C01803=1094.320,109.025,-62.367,176.115,17.436,152.491
C01804=1094.315,108.775,-62.348,176.112,17.435,152.491
C01805=1094.309,108.526,-62.329,176.109,17.434,152.491
C01806=1094.303,108.277,-62.310,176.107,17.434,152.491
C01807=1094.297,108.028,-62.292,176.104,17.433,152.492
C01808=1094.292,107.779,-62.274,176.102,17.431,152.492
C01809=1094.287,107.529,-62.254,176.100,17.431,152.492
C01810=1094.280,107.279,-62.236,176.097,17.430,152.493
C01811=1094.275,107.031,-62.218,176.095,17.429,152.493
C01812=1094.269,106.782,-62.199,176.092,17.428,152.493
C01813=1094.264,106.532,-62.181,176.089,17.428,152.494
C01814=1094.258,106.283,-62.162,176.087,17.427,152.494
C01815=1094.253,106.034,-62.144,176.085,17.426,152.494
C01816=1094.247,105.785,-62.125,176.082,17.424,152.494
C01817=1094.241,105.535,-62.106,176.080,17.424,152.495
C01818=1094.236,105.286,-62.088,176.077,17.423,152.495
C01819=1094.230,105.037,-62.069,176.075,17.422,152.495
C01820=1094.225,104.787,-62.051,176.072,17.421,152.496
C01821=1094.218,104.538,-62.032,176.070,17.420,152.496
C01822=1094.214,104.289,-62.014,176.067,17.420,152.496
C01823=1094.207,104.040,-61.996,176.065,17.419,152.497
C01824=1094.202,103.790,-61.978,176.063,17.418,152.497
C01825=1094.196,103.541,-61.959,176.060,17.417,152.497
C01826=1094.191,103.292,-61.941,176.057,17.416,152.497
C01827=1094.185,103.043,-61.922,176.055,17.415,152.498
C01828=1094.180,102.794,-61.904,176.053,17.414,152.498
C01829=1094.174,102.544,-61.885,176.050,17.413,152.498
C01830=1094.169,102.295,-61.867,176.048,17.412,152.498
C01831=1094.162,102.046,-61.848,176.045,17.411,152.499
C01832=1094.158,101.797,-61.830,176.043,17.411,152.499
C01833=1094.152,101.547,-61.812,176.040,17.409,152.499
C01834=1094.146,101.298,-61.793,176.038,17.408,152.500
C01835=1094.140,101.048,-61.776,176.036,17.408,152.500
C01836=1094.134,100.800,-61.757,176.033,17.407,152.500
C01837=1094.129,100.550,-61.739,176.031,17.406,152.500
C01838=1094.124,100.301,-61.721,176.028,17.405,152.501
C01839=1094.117,100.052,-61.702,176.026,17.404,152.501
C01840=1094.112,99.802,-61.684,176.024,17.403,152.501
C01841=1094.106,99.553,-61.666,176.021,17.402,152.501
C01842=1094.100,99.304,-61.648,176.019,17.401,152.502
C01843=1094.095,99.054,-61.630,176.016,17.401,152.502
C01844=1094.090,98.805,-61.612,176.014,17.400,152.502
C01845=1094.083,98.556,-61.593,176.011,17.399,152.503
C01846=1094.078,98.307,-61.575,176.009,17.397,152.503
C01847=1094.072,98.057,-61.557,176.007,17.397,152.503
C01848=1094.066,97.809,-61.539,176.004,17.396,152.503
C01849=1094.060,97.559,-61.521,176.002,17.395,152.504
C01850=1094.055,97.309,-61.503,175.999,17.394,152.504
C01851=1094.049,97.060,-61.485,175.997,17.393,152.504
C01852=1094.044,96.811,-61.467,175.995,17.392,152.504
C01853=1094.039,96.562,-61.449,175.992,17.391,152.505
C01854=1094.033,96.312,-61.431,175.990,17.390,152.505
C01855=1094.026,96.037,-61.411,175.987,17.389,152.505
C01856=1094.020,95.761,-61.392,175.984,17.388,152.506
C01857=1094.014,95.485,-61.370,175.982,17.387,152.506
C01858=1094.008,95.210,-61.351,175.979,17.386,152.506
C01859=1094.002,94.961,-61.333,175.977,17.385,152.507
C01860=1093.996,94.711,-61.315,175.974,17.384,152.507
C01861=1093.991,94.462,-61.297,175.973,17.383,152.507
C01862=1093.985,94.213,-61.279,175.970,17.382,152.507
C01863=1093.979,93.963,-61.261,175.967,17.381,152.508
C01864=1093.974,93.714,-61.243,175.965,17.380,152.508
C01865=1093.969,93.465,-61.225,175.962,17.379,152.508
C01866=1093.963,93.215,-61.207,175.961,17.378,152.508
C01867=1093.957,92.966,-61.190,175.958,17.377,152.508
C01868=1093.951,92.716,-61.172,175.955,17.376,152.509
C01869=1093.946,92.467,-61.154,175.954,17.375,152.509
C01870=1093.941,92.218,-61.136,175.951,17.374,152.509
C01871=1093.935,91.968,-61.118,175.949,17.373,152.509
C01872=1093.929,91.719,-61.101,175.946,17.372,152.510
C01873=1093.923,91.471,-61.082,175.944,17.371,152.510
C01874=1093.917,91.221,-61.064,175.942,17.370,152.510
C01875=1093.912,90.972,-61.046,175.939,17.369,152.511
C01876=1093.907,90.723,-61.029,175.937,17.368,152.511
C01877=1093.901,90.473,-61.011,175.934,17.367,152.511
C01878=1093.895,90.224,-60.993,175.932,17.366,152.511
C01879=1093.890,89.975,-60.976,175.930,17.365,152.512
C01880=1093.884,89.725,-60.958,175.928,17.364,152.512
C01881=1093.878,89.476,-60.940,175.925,17.363,152.512
C01882=1093.873,89.227,-60.922,175.923,17.362,152.512
C01883=1093.866,88.977,-60.905,175.921,17.361,152.512
C01884=1093.861,88.728,-60.887,175.918,17.360,152.513
C01885=1093.856,88.479,-60.870,175.916,17.359,152.513
C01886=1093.850,88.229,-60.852,175.913,17.358,152.513
C01887=1093.844,87.980,-60.835,175.911,17.357,152.514
C01888=1093.839,87.731,-60.817,175.909,17.356,152.514
C01889=1093.832,87.481,-60.799,175.907,17.355,152.514
C01890=1093.827,87.232,-60.782,175.904,17.354,152.514
C01891=1093.821,86.983,-60.764,175.902,17.353,152.514
C01892=1093.815,86.733,-60.746,175.900,17.352,152.515
C01893=1093.810,86.484,-60.728,175.897,17.351,152.515
C01894=1093.804,86.235,-60.711,175.895,17.350,152.515
C01895=1093.798,85.985,-60.694,175.892,17.349,152.515
C01896=1093.793,85.736,-60.676,175.891,17.348,152.516
C01897=1093.787,85.487,-60.659,175.888,17.347,152.516
C01898=1093.781,85.238,-60.642,175.886,17.346,152.516
C01899=1093.775,84.988,-60.624,175.883,17.345,152.516
C01900=1093.770,84.739,-60.606,175.881,17.344,152.517
C01901=1093.764,84.490,-60.589,175.879,17.342,152.517
C01902=1093.759,84.241,-60.572,175.877,17.342,152.517
C01903=1093.753,83.991,-60.554,175.874,17.341,152.517
C01904=1093.747,83.742,-60.536,175.872,17.339,152.518
C01905=1093.742,83.492,-60.519,175.870,17.338,152.518
C01906=1093.736,83.243,-60.502,175.867,17.337,152.518
C01907=1093.730,82.993,-60.484,175.865,17.336,152.518
C01908=1093.725,82.744,-60.466,175.863,17.335,152.518
C01909=1093.720,82.495,-60.449,175.861,17.334,152.519
C01910=1093.714,82.246,-60.432,175.858,17.333,152.519
C01911=1093.708,81.997,-60.415,175.856,17.332,152.519
C01912=1093.702,81.746,-60.398,175.854,17.331,152.519
C01913=1093.696,81.497,-60.380,175.852,17.330,152.519
C01914=1093.691,81.248,-60.363,175.849,17.329,152.520
C01915=1093.685,80.999,-60.345,175.847,17.328,152.520
C01916=1093.680,80.750,-60.328,175.845,17.326,152.520
C01917=1093.675,80.501,-60.311,175.842,17.325,152.520
C01918=1093.669,80.250,-60.293,175.840,17.325,152.521
C01919=1093.662,79.975,-60.274,175.838,17.323,152.521
C01920=1093.656,79.700,-60.255,175.835,17.322,152.521
C01921=1093.650,79.424,-60.236,175.833,17.321,152.521
C01922=1093.644,79.149,-60.217,175.831,17.319,152.521
C01923=1093.639,78.900,-60.199,175.828,17.318,152.522
C01924=1093.633,78.650,-60.183,175.826,17.318,152.522
C01925=1093.627,78.400,-60.165,175.824,17.316,152.522
C01926=1093.621,78.151,-60.148,175.822,17.315,152.522
C01927=1093.616,77.902,-60.131,175.819,17.314,152.523
C01928=1093.610,77.652,-60.114,175.818,17.313,152.523
C01929=1093.604,77.403,-60.097,175.815,17.312,152.523
C01930=1093.599,77.154,-60.080,175.813,17.311,152.523
C01931=1093.592,76.904,-60.063,175.811,17.309,152.523
C01932=1093.587,76.655,-60.045,175.809,17.309,152.524
C01933=1093.582,76.406,-60.028,175.806,17.308,152.524
C01934=1093.576,76.157,-60.011,175.803,17.306,152.524
C01935=1093.570,75.907,-59.994,175.802,17.305,152.524
C01936=1093.565,75.658,-59.977,175.799,17.304,152.524
C01937=1093.559,75.409,-59.960,175.797,17.303,152.525
C01938=1093.553,75.158,-59.943,175.795,17.302,152.525
C01939=1093.547,74.909,-59.926,175.793,17.301,152.525
C01940=1093.541,74.660,-59.910,175.790,17.299,152.525
C01941=1093.536,74.411,-59.892,175.789,17.298,152.525
C01942=1093.531,74.161,-59.875,175.786,17.297,152.526
C01943=1093.524,73.913,-59.858,175.784,17.296,152.526
C01944=1093.519,73.663,-59.841,175.781,17.295,152.526
C01945=1093.514,73.414,-59.824,175.780,17.294,152.526
C01946=1093.508,73.165,-59.808,175.777,17.292,152.526
C01947=1093.502,72.914,-59.790,175.775,17.292,152.527
C01948=1093.496,72.665,-59.773,175.773,17.290,152.527
C01949=1093.490,72.416,-59.757,175.771,17.289,152.527
C01950=1093.485,72.166,-59.740,175.768,17.288,152.527
C01951=1093.479,71.917,-59.723,175.767,17.287,152.527
C01952=1093.474,71.668,-59.706,175.764,17.286,152.528
C01953=1093.468,71.418,-59.689,175.762,17.285,152.528
C01954=1093.462,71.169,-59.672,175.759,17.284,152.528
C01955=1093.457,70.920,-59.655,175.758,17.283,152.528
C01956=1093.451,70.670,-59.639,175.755,17.281,152.528
C01957=1093.446,70.421,-59.621,175.753,17.280,152.528
C01958=1093.440,70.172,-59.605,175.751,17.279,152.529
C01959=1093.434,69.922,-59.588,175.749,17.278,152.529
C01960=1093.429,69.673,-59.571,175.746,17.277,152.529
C01961=1093.423,69.424,-59.554,175.745,17.276,152.529
C01962=1093.417,69.175,-59.538,175.742,17.274,152.529
C01963=1093.412,68.925,-59.521,175.740,17.273,152.530
C01964=1093.405,68.676,-59.504,175.738,17.272,152.530
C01965=1093.400,68.426,-59.487,175.736,17.271,152.530
C01966=1093.394,68.177,-59.471,175.734,17.269,152.530
C01967=1093.388,67.927,-59.454,175.732,17.269,152.530
C01968=1093.383,67.677,-59.438,175.729,17.267,152.530
C01969=1093.377,67.428,-59.420,175.727,17.266,152.531
C01970=1093.371,67.179,-59.404,175.725,17.265,152.531
C01971=1093.366,66.929,-59.387,175.723,17.264,152.531
C01972=1093.360,66.680,-59.371,175.721,17.262,152.531
C01973=1093.355,66.430,-59.354,175.719,17.262,152.531
C01974=1093.348,66.182,-59.337,175.716,17.260,152.532
C01975=1093.342,65.932,-59.321,175.714,17.259,152.532
C01976=1093.337,65.683,-59.304,175.712,17.258,152.532
C01977=1093.331,65.433,-59.288,175.710,17.257,152.532
C01978=1093.326,65.184,-59.271,175.708,17.256,152.532
C01979=1093.320,64.934,-59.255,175.706,17.254,152.532
C01980=1093.314,64.685,-59.238,175.704,17.254,152.533
C01981=1093.309,64.435,-59.221,175.702,17.252,152.533
C01982=1093.303,64.186,-59.205,175.700,17.251,152.533
C01983=1093.297,63.911,-59.187,175.697,17.250,152.533
C01984=1093.290,63.636,-59.168,175.695,17.248,152.533
C01985=1093.283,63.360,-59.150,175.692,17.247,152.534
C01986=1093.277,63.085,-59.132,175.690,17.246,152.534
C01987=1093.272,62.835,-59.115,175.688,17.244,152.534
C01988=1093.266,62.586,-59.099,175.686,17.243,152.534
C01989=1093.260,62.336,-59.083,175.683,17.242,152.534
C01990=1093.254,62.087,-59.067,175.682,17.241,152.534
C01991=1093.249,61.837,-59.050,175.679,17.240,152.535
C01992=1093.243,61.588,-59.034,175.677,17.239,152.535
C01993=1093.237,61.339,-59.017,175.675,17.237,152.535
C01994=1093.231,61.089,-59.001,175.673,17.236,152.535
C01995=1093.225,60.840,-58.985,175.671,17.235,152.535
C01996=1093.220,60.590,-58.968,175.669,17.234,152.535
C01997=1093.214,60.341,-58.952,175.667,17.233,152.536
C01998=1093.208,60.092,-58.935,175.664,17.232,152.536
C01999=1093.202,59.842,-58.920,175.663,17.231,152.536
C02000=1093.196,59.592,-58.904,175.660,17.229,152.536
C02001=1093.191,59.343,-58.887,175.658,17.228,152.536
C02002=1093.185,59.093,-58.871,175.656,17.227,152.536
C02003=1093.179,58.844,-58.854,175.654,17.225,152.537
C02004=1093.173,58.595,-58.838,175.652,17.224,152.537
C02005=1093.167,58.345,-58.822,175.650,17.223,152.537
C02006=1093.162,58.096,-58.806,175.648,17.221,152.537
C02007=1093.156,57.846,-58.789,175.646,17.221,152.537
C02008=1093.151,57.598,-58.773,175.644,17.220,152.537
C02009=1093.145,57.348,-58.757,175.642,17.218,152.538
C02010=1093.139,57.098,-58.741,175.640,17.217,152.538
C02011=1093.133,56.849,-58.725,175.637,17.216,152.538
C02012=1093.127,56.600,-58.708,175.636,17.215,152.538
C02013=1093.121,56.350,-58.692,175.633,17.213,152.538
C02014=1093.116,56.101,-58.676,175.631,17.212,152.538
C02015=1093.111,55.851,-58.660,175.629,17.211,152.539
C02016=1093.105,55.602,-58.644,175.627,17.209,152.539
C02017=1093.099,55.353,-58.628,175.625,17.209,152.539
C02018=1093.093,55.103,-58.611,175.623,17.207,152.539
C02019=1093.087,54.854,-58.595,175.621,17.206,152.539
C02020=1093.082,54.604,-58.580,175.619,17.204,152.539
C02021=1093.076,54.355,-58.563,175.617,17.204,152.539
C02022=1093.070,54.105,-58.547,175.614,17.202,152.540
C02023=1093.065,53.857,-58.531,175.613,17.201,152.540
C02024=1093.059,53.607,-58.516,175.610,17.199,152.540
C02025=1093.054,53.357,-58.499,175.608,17.199,152.540
C02026=1093.048,53.108,-58.483,175.607,17.197,152.540
C02027=1093.042,52.858,-58.467,175.604,17.196,152.540
C02028=1093.037,52.609,-58.451,175.603,17.195,152.540
C02029=1093.031,52.360,-58.435,175.600,17.193,152.541
C02030=1093.025,52.110,-58.419,175.598,17.192,152.541
C02031=1093.019,51.860,-58.403,175.596,17.191,152.541
C02032=1093.013,51.611,-58.387,175.594,17.190,152.541
C02033=1093.008,51.362,-58.372,175.592,17.188,152.541
C02034=1093.002,51.112,-58.355,175.590,17.187,152.541
C02035=1092.996,50.863,-58.339,175.589,17.186,152.541
C02036=1092.991,50.613,-58.324,175.586,17.184,152.542
C02037=1092.985,50.364,-58.308,175.584,17.183,152.542
C02038=1092.979,50.115,-58.291,175.582,17.182,152.542
C02039=1092.974,49.865,-58.276,175.580,17.181,152.542
C02040=1092.968,49.616,-58.260,175.578,17.179,152.542
C02041=1092.963,49.366,-58.244,175.576,17.178,152.542
C02042=1092.957,49.117,-58.228,175.575,17.177,152.542
C02043=1092.951,48.868,-58.212,175.572,17.175,152.543
C02044=1092.945,48.618,-58.196,175.570,17.174,152.543
C02045=1092.940,48.369,-58.181,175.568,17.173,152.543
C02046=1092.934,48.119,-58.165,175.566,17.171,152.543
C02047=1092.928,47.843,-58.147,175.564,17.170,152.543
C02048=1092.922,47.568,-58.130,175.561,17.168,152.543
C02049=1092.915,47.291,-58.112,175.560,17.167,152.543
C02050=1092.910,47.015,-58.095,175.557,17.165,152.543
C02051=1092.904,46.766,-58.079,175.556,17.164,152.543
C02052=1092.899,46.517,-58.064,175.553,17.163,152.544
C02053=1092.893,46.267,-58.047,175.551,17.161,152.544
C02054=1092.887,46.017,-58.032,175.549,17.160,152.544
C02055=1092.882,45.769,-58.016,175.547,17.159,152.544
C02056=1092.876,45.519,-58.000,175.546,17.158,152.544
C02057=1092.870,45.269,-57.984,175.543,17.156,152.544
C02058=1092.865,45.020,-57.969,175.541,17.155,152.544
C02059=1092.859,44.770,-57.953,175.539,17.153,152.544
C02060=1092.853,44.521,-57.937,175.537,17.152,152.545
C02061=1092.848,44.272,-57.922,175.535,17.151,152.545
C02062=1092.842,44.022,-57.906,175.533,17.150,152.545
C02063=1092.837,43.772,-57.890,175.532,17.148,152.545
C02064=1092.831,43.523,-57.876,175.529,17.147,152.545
C02065=1092.825,43.274,-57.859,175.528,17.146,152.545
C02066=1092.819,43.024,-57.844,175.525,17.144,152.545
C02067=1092.814,42.775,-57.828,175.524,17.143,152.545
C02068=1092.808,42.525,-57.812,175.522,17.142,152.545
C02069=1092.802,42.276,-57.797,175.519,17.140,152.546
C02070=1092.797,42.027,-57.782,175.518,17.139,152.546
C02071=1092.791,41.777,-57.766,175.515,17.137,152.546
C02072=1092.785,41.527,-57.750,175.514,17.136,152.546
C02073=1092.779,41.279,-57.735,175.512,17.135,152.546
C02074=1092.774,41.029,-57.720,175.510,17.133,152.546
C02075=1092.768,40.779,-57.704,175.508,17.133,152.546
C02076=1092.763,40.530,-57.688,175.505,17.131,152.547
C02077=1092.756,40.281,-57.673,175.504,17.130,152.547
C02078=1092.751,40.031,-57.658,175.502,17.129,152.547
C02079=1092.746,39.781,-57.642,175.500,17.127,152.547
C02080=1092.740,39.532,-57.626,175.498,17.126,152.547
C02081=1092.734,39.283,-57.612,175.496,17.124,152.547
C02082=1092.728,39.033,-57.596,175.494,17.123,152.547
C02083=1092.723,38.783,-57.581,175.492,17.122,152.547
C02084=1092.717,38.534,-57.565,175.490,17.120,152.547
C02085=1092.711,38.285,-57.550,175.488,17.119,152.547
C02086=1092.706,38.036,-57.535,175.486,17.118,152.548
C02087=1092.700,37.786,-57.519,175.484,17.116,152.548
C02088=1092.694,37.536,-57.504,175.483,17.115,152.548
C02089=1092.688,37.287,-57.488,175.480,17.114,152.548
C02090=1092.683,37.037,-57.473,175.479,17.112,152.548
C02091=1092.677,36.788,-57.458,175.477,17.111,152.548
C02092=1092.671,36.538,-57.443,175.474,17.110,152.548
C02093=1092.665,36.289,-57.428,175.473,17.109,152.548
C02094=1092.660,36.039,-57.412,175.470,17.107,152.549
C02095=1092.653,35.790,-57.397,175.469,17.106,152.549
C02096=1092.648,35.540,-57.381,175.467,17.105,152.549
C02097=1092.643,35.291,-57.366,175.465,17.103,152.549
C02098=1092.636,35.042,-57.351,175.463,17.102,152.549
C02099=1092.631,34.792,-57.336,175.461,17.100,152.549
C02100=1092.625,34.543,-57.321,175.459,17.099,152.549
C02101=1092.620,34.293,-57.306,175.457,17.098,152.549
C02102=1092.613,34.044,-57.291,175.455,17.096,152.549
C02103=1092.608,33.794,-57.275,175.453,17.095,152.549
C02104=1092.602,33.545,-57.260,175.452,17.094,152.550
C02105=1092.596,33.295,-57.244,175.449,17.092,152.550
C02106=1092.591,33.046,-57.229,175.448,17.091,152.550
C02107=1092.585,32.796,-57.214,175.446,17.090,152.550
C02108=1092.579,32.547,-57.199,175.444,17.088,152.550
C02109=1092.573,32.298,-57.184,175.442,17.087,152.550
C02110=1092.568,32.048,-57.169,175.440,17.085,152.550
C02111=1092.561,31.772,-57.152,175.438,17.084,152.550
C02112=1092.555,31.496,-57.136,175.436,17.082,152.550
C02113=1092.549,31.220,-57.119,175.434,17.081,152.550
C02114=1092.542,30.945,-57.103,175.432,17.079,152.551
C02115=1092.537,30.695,-57.087,175.430,17.078,152.551
C02116=1092.531,30.446,-57.073,175.428,17.077,152.551
C02117=1092.525,30.196,-57.057,175.426,17.076,152.551
C02118=1092.520,29.947,-57.042,175.424,17.074,152.551
C02119=1092.514,29.697,-57.027,175.422,17.072,152.551
C02120=1092.508,29.448,-57.012,175.421,17.071,152.551
C02121=1092.503,29.198,-56.997,175.418,17.069,152.551
C02122=1092.497,28.949,-56.983,175.416,17.068,152.551
C02123=1092.491,28.699,-56.968,175.415,17.067,152.551
C02124=1092.486,28.450,-56.953,175.412,17.066,152.552
C02125=1092.479,28.200,-56.938,175.411,17.064,152.552
C02126=1092.474,27.951,-56.923,175.409,17.063,152.552
C02127=1092.468,27.701,-56.908,175.407,17.062,152.552
C02128=1092.462,27.452,-56.893,175.405,17.060,152.552
C02129=1092.456,27.202,-56.878,175.403,17.059,152.552
C02130=1092.451,26.953,-56.863,175.401,17.057,152.552
C02131=1092.445,26.703,-56.849,175.400,17.056,152.552
C02132=1092.440,26.454,-56.834,175.398,17.055,152.552
C02133=1092.433,26.204,-56.819,175.396,17.053,152.552
C02134=1092.427,25.955,-56.804,175.394,17.052,152.553
C02135=1092.422,25.705,-56.789,175.392,17.051,152.553
C02136=1092.416,25.456,-56.774,175.390,17.049,152.553
C02137=1092.410,25.206,-56.760,175.388,17.048,152.553
C02138=1092.405,24.957,-56.745,175.387,17.047,152.553
C02139=1092.399,24.708,-56.730,175.385,17.045,152.553
C02140=1092.393,24.458,-56.715,175.383,17.044,152.553
C02141=1092.388,24.208,-56.701,175.380,17.042,152.553
C02142=1092.382,23.958,-56.686,175.379,17.041,152.553
C02143=1092.376,23.709,-56.671,175.377,17.040,152.553
C02144=1092.369,23.460,-56.656,175.375,17.038,152.553
C02145=1092.365,23.210,-56.642,175.373,17.037,152.554
C02146=1092.359,22.961,-56.627,175.372,17.035,152.554
C02147=1092.352,22.711,-56.612,175.369,17.034,152.554
C02148=1092.347,22.462,-56.597,175.368,17.033,152.554
C02149=1092.341,22.212,-56.583,175.366,17.032,152.554
C02150=1092.336,21.963,-56.568,175.364,17.030,152.554
C02151=1092.329,21.713,-56.553,175.362,17.029,152.554
C02152=1092.324,21.463,-56.539,175.360,17.028,152.554
C02153=1092.319,21.214,-56.524,175.358,17.025,152.554
C02154=1092.312,20.965,-56.509,175.357,17.024,152.554
C02155=1092.307,20.715,-56.495,175.355,17.023,152.554
C02156=1092.302,20.466,-56.480,175.353,17.022,152.554
C02157=1092.295,20.216,-56.465,175.351,17.020,152.555
C02158=1092.290,19.967,-56.451,175.350,17.019,152.555
C02159=1092.284,19.717,-56.436,175.348,17.018,152.555
C02160=1092.278,19.468,-56.422,175.346,17.016,152.555
C02161=1092.272,19.218,-56.408,175.344,17.015,152.555
C02162=1092.267,18.968,-56.392,175.342,17.014,152.555
C02163=1092.261,18.719,-56.379,175.340,17.012,152.555
C02164=1092.255,18.469,-56.364,175.339,17.010,152.555
C02165=1092.249,18.220,-56.349,175.337,17.009,152.555
C02166=1092.243,17.971,-56.335,175.334,17.008,152.555
C02167=1092.237,17.721,-56.320,175.333,17.006,152.555
C02168=1092.232,17.471,-56.306,175.331,17.005,152.555
C02169=1092.227,17.222,-56.291,175.329,17.004,152.556
C02170=1092.221,16.972,-56.277,175.327,17.002,152.556
C02171=1092.215,16.723,-56.262,175.326,17.001,152.556
C02172=1092.209,16.473,-56.248,175.323,16.999,152.556
C02173=1092.203,16.224,-56.234,175.322,16.998,152.556
C02174=1092.197,15.975,-56.219,175.320,16.997,152.556
C02175=1092.191,15.700,-56.203,175.318,16.995,152.556
C02176=1092.185,15.426,-56.187,175.316,16.994,152.556
C02177=1092.178,15.151,-56.172,175.314,16.992,152.556
C02178=1092.172,14.876,-56.155,175.312,16.991,152.556
C02179=1092.167,14.627,-56.142,175.310,16.989,152.556
C02180=1092.161,14.378,-56.127,175.308,16.988,152.556
C02181=1092.155,14.128,-56.113,175.307,16.986,152.557
C02182=1092.149,13.879,-56.098,175.304,16.985,152.557
C02183=1092.143,13.629,-56.084,175.303,16.984,152.557
C02184=1092.137,13.379,-56.070,175.301,16.982,152.557
C02185=1092.132,13.130,-56.056,175.300,16.981,152.557
C02186=1092.126,12.880,-56.042,175.297,16.979,152.557
C02187=1092.120,12.631,-56.027,175.296,16.978,152.557
C02188=1092.113,12.381,-56.013,175.294,16.977,152.557
C02189=1092.108,12.132,-55.999,175.292,16.975,152.557
C02190=1092.102,11.882,-55.985,175.290,16.974,152.557
C02191=1092.096,11.633,-55.971,175.289,16.973,152.557
C02192=1092.090,11.384,-55.956,175.287,16.971,152.557
C02193=1092.084,11.133,-55.942,175.285,16.970,152.558
C02194=1092.079,10.884,-55.928,175.283,16.969,152.558
C02195=1092.073,10.635,-55.914,175.282,16.967,152.558
C02196=1092.067,10.385,-55.899,175.279,16.965,152.558
C02197=1092.061,10.135,-55.885,175.278,16.964,152.558
C02198=1092.056,9.886,-55.871,175.276,16.963,152.558
C02199=1092.049,9.637,-55.858,175.274,16.962,152.558
C02200=1092.043,9.386,-55.843,175.272,16.960,152.558
C02201=1092.038,9.138,-55.829,175.271,16.959,152.558
C02202=1092.032,8.888,-55.815,175.269,16.958,152.558
C02203=1092.027,8.638,-55.801,175.267,16.956,152.558
C02204=1092.020,8.389,-55.786,175.265,16.954,152.558
C02205=1092.015,8.139,-55.772,175.264,16.953,152.558
C02206=1092.009,7.890,-55.758,175.262,16.952,152.558
C02207=1092.003,7.640,-55.745,175.260,16.950,152.559
C02208=1091.997,7.391,-55.730,175.258,16.949,152.559
C02209=1091.991,7.141,-55.716,175.257,16.948,152.559
C02210=1091.986,6.892,-55.702,175.254,16.946,152.559
C02211=1091.980,6.642,-55.689,175.252,16.945,152.559
C02212=1091.974,6.392,-55.674,175.251,16.943,152.559
C02213=1091.968,6.143,-55.660,175.250,16.942,152.559
C02214=1091.962,5.893,-55.646,175.247,16.940,152.559
C02215=1091.957,5.644,-55.633,175.245,16.939,152.559
C02216=1091.951,5.394,-55.619,175.244,16.938,152.559
C02217=1091.945,5.145,-55.604,175.242,16.937,152.559
C02218=1091.939,4.895,-55.590,175.240,16.935,152.559
C02219=1091.933,4.646,-55.577,175.238,16.934,152.559
C02220=1091.928,4.396,-55.563,175.237,16.932,152.559
C02221=1091.922,4.147,-55.549,175.235,16.930,152.560
C02222=1091.916,3.896,-55.535,175.233,16.929,152.560
C02223=1091.910,3.647,-55.520,175.232,16.928,152.560
C02224=1091.904,3.398,-55.507,175.230,16.927,152.560
C02225=1091.899,3.149,-55.493,175.228,16.925,152.560
C02226=1091.893,2.899,-55.479,175.226,16.924,152.560
C02227=1091.888,2.649,-55.465,175.225,16.922,152.560
C02228=1091.882,2.400,-55.451,175.223,16.921,152.560
C02229=1091.875,2.150,-55.438,175.221,16.919,152.560
C02230=1091.870,1.900,-55.424,175.219,16.918,152.560
C02231=1091.865,1.651,-55.410,175.218,16.917,152.560
C02232=1091.859,1.401,-55.396,175.216,16.915,152.560
C02233=1091.854,1.152,-55.382,175.214,16.913,152.560
C02234=1091.847,0.902,-55.369,175.212,16.912,152.560
C02235=1091.842,0.653,-55.354,175.211,16.911,152.560
C02236=1091.836,0.404,-55.341,175.209,16.909,152.560
C02237=1091.830,0.154,-55.326,175.207,16.908,152.561
C02238=1091.824,-0.096,-55.313,175.205,16.907,152.561
C02239=1091.818,-0.369,-55.298,175.204,16.905,152.561
C02240=1091.812,-0.641,-55.283,175.201,16.903,152.561
C02241=1091.805,-0.913,-55.268,175.200,16.902,152.561
C02242=1091.800,-1.186,-55.253,175.198,16.900,152.561
C02243=1091.794,-1.435,-55.240,175.196,16.899,152.561
C02244=1091.788,-1.685,-55.226,175.194,16.898,152.561
C02245=1091.782,-1.935,-55.212,175.192,16.896,152.561
C02246=1091.777,-2.185,-55.198,175.191,16.894,152.561
C02247=1091.770,-2.434,-55.185,175.189,16.893,152.561
C02248=1091.765,-2.683,-55.171,175.188,16.892,152.561
C02249=1091.760,-2.933,-55.157,175.185,16.890,152.561
C02250=1091.753,-3.182,-55.144,175.184,16.889,152.561
C02251=1091.748,-3.432,-55.130,175.182,16.887,152.561
C02252=1091.742,-3.681,-55.116,175.181,16.886,152.561
C02253=1091.736,-3.931,-55.103,175.179,16.885,152.562
C02254=1091.731,-4.180,-55.089,175.177,16.883,152.562
C02255=1091.725,-4.430,-55.077,175.175,16.882,152.562
C02256=1091.719,-4.680,-55.062,175.174,16.881,152.562
C02257=1091.712,-4.930,-55.049,175.172,16.880,152.562
C02258=1091.707,-5.179,-55.035,175.170,16.877,152.562
C02259=1091.701,-5.428,-55.022,175.168,16.876,152.562
C02260=1091.695,-5.678,-55.008,175.167,16.875,152.562
C02261=1091.689,-5.927,-54.995,175.165,16.874,152.562
C02262=1091.684,-6.177,-54.981,175.163,16.872,152.562
C02263=1091.678,-6.427,-54.968,175.161,16.871,152.562
C02264=1091.672,-6.676,-54.955,175.160,16.870,152.562
C02265=1091.666,-6.926,-54.941,175.158,16.868,152.562
C02266=1091.661,-7.175,-54.927,175.157,16.867,152.562
C02267=1091.654,-7.424,-54.914,175.154,16.865,152.563
C02268=1091.649,-7.675,-54.901,175.153,16.864,152.563
C02269=1091.642,-7.925,-54.887,175.151,16.862,152.563
C02270=1091.637,-8.174,-54.873,175.150,16.861,152.563
C02271=1091.631,-8.423,-54.860,175.147,16.860,152.563
C02272=1091.624,-8.673,-54.847,175.146,16.858,152.563
C02273=1091.619,-8.923,-54.834,175.144,16.857,152.563
C02274=1091.613,-9.172,-54.821,175.143,16.856,152.563
C02275=1091.608,-9.422,-54.807,175.141,16.854,152.563
C02276=1091.601,-9.671,-54.793,175.139,16.852,152.563
C02277=1091.596,-9.921,-54.780,175.137,16.851,152.563
C02278=1091.590,-10.170,-54.767,175.136,16.850,152.563
C02279=1091.584,-10.420,-54.753,175.134,16.849,152.563
C02280=1091.579,-10.670,-54.741,175.133,16.847,152.563
C02281=1091.572,-10.919,-54.727,175.130,16.845,152.563
C02282=1091.567,-11.169,-54.713,175.129,16.844,152.563
C02283=1091.561,-11.418,-54.700,175.127,16.843,152.563
C02284=1091.556,-11.668,-54.687,175.126,16.842,152.564
C02285=1091.549,-11.917,-54.674,175.123,16.840,152.564
C02286=1091.544,-12.167,-54.660,175.122,16.839,152.564
C02287=1091.538,-12.417,-54.647,175.120,16.837,152.564
C02288=1091.532,-12.666,-54.634,175.119,16.836,152.564
C02289=1091.527,-12.916,-54.621,175.117,16.835,152.564
C02290=1091.520,-13.166,-54.608,175.115,16.833,152.564
C02291=1091.515,-13.415,-54.594,175.113,16.831,152.564
C02292=1091.510,-13.664,-54.582,175.112,16.830,152.564
C02293=1091.503,-13.914,-54.568,175.110,16.829,152.564
C02294=1091.498,-14.163,-54.554,175.109,16.828,152.564
C02295=1091.492,-14.413,-54.542,175.106,16.826,152.564
C02296=1091.486,-14.663,-54.528,175.105,16.824,152.564
C02297=1091.481,-14.913,-54.515,175.103,16.823,152.564
C02298=1091.474,-15.162,-54.502,175.102,16.822,152.564
C02299=1091.469,-15.412,-54.489,175.100,16.821,152.564
C02300=1091.463,-15.661,-54.476,175.098,16.819,152.564
C02301=1091.457,-15.911,-54.462,175.096,16.818,152.565
C02302=1091.451,-16.160,-54.450,175.095,16.816,152.565
C02303=1091.444,-16.431,-54.436,175.093,16.815,152.565
C02304=1091.438,-16.702,-54.421,175.091,16.813,152.565
C02305=1091.432,-16.972,-54.407,175.089,16.812,152.565
C02306=1091.425,-17.243,-54.393,175.088,16.810,152.565
C02307=1091.419,-17.493,-54.380,175.086,16.809,152.565
C02308=1091.413,-17.743,-54.367,175.084,16.808,152.565
C02309=1091.408,-17.993,-54.354,175.082,16.806,152.565
C02310=1091.402,-18.242,-54.341,175.081,16.805,152.565
C02311=1091.396,-18.492,-54.328,175.079,16.804,152.565
C02312=1091.390,-18.741,-54.315,175.078,16.803,152.565
C02313=1091.384,-18.991,-54.302,175.076,16.800,152.565
C02314=1091.378,-19.241,-54.289,175.074,16.799,152.565
C02315=1091.373,-19.490,-54.276,175.072,16.798,152.566
C02316=1091.367,-19.739,-54.263,175.071,16.797,152.565
C02317=1091.361,-19.989,-54.250,175.069,16.795,152.566
C02318=1091.355,-20.238,-54.237,175.067,16.794,152.566
C02319=1091.350,-20.488,-54.224,175.065,16.793,152.566
C02320=1091.344,-20.738,-54.212,175.064,16.791,152.566
C02321=1091.337,-20.988,-54.198,175.062,16.790,152.566
C02322=1091.331,-21.237,-54.186,175.061,16.789,152.566
C02323=1091.325,-21.487,-54.172,175.059,16.787,152.566
C02324=1091.319,-21.737,-54.160,175.057,16.785,152.566
C02325=1091.315,-21.986,-54.147,175.055,16.784,152.566
C02326=1091.309,-22.235,-54.134,175.054,16.783,152.566
C02327=1091.303,-22.485,-54.121,175.052,16.782,152.566
C02328=1091.297,-22.735,-54.109,175.051,16.780,152.566
C02329=1091.291,-22.984,-54.095,175.049,16.779,152.566
C02330=1091.285,-23.234,-54.083,175.047,16.777,152.566
C02331=1091.279,-23.484,-54.070,175.045,16.776,152.566
C02332=1091.274,-23.733,-54.057,175.044,16.775,152.567
C02333=1091.268,-23.983,-54.044,175.042,16.773,152.567
C02334=1091.262,-24.233,-54.032,175.041,16.772,152.567
C02335=1091.256,-24.482,-54.018,175.039,16.771,152.567
C02336=1091.250,-24.732,-54.006,175.037,16.769,152.567
C02337=1091.245,-24.981,-53.994,175.035,16.768,152.567
C02338=1091.238,-25.230,-53.980,175.034,16.767,152.567
C02339=1091.232,-25.480,-53.968,175.032,16.765,152.567
C02340=1091.227,-25.730,-53.955,175.031,16.764,152.567
C02341=1091.221,-25.980,-53.942,175.029,16.763,152.567
C02342=1091.216,-26.229,-53.929,175.028,16.761,152.567
C02343=1091.210,-26.479,-53.917,175.025,16.759,152.567
C02344=1091.204,-26.729,-53.904,175.024,16.758,152.567
C02345=1091.198,-26.979,-53.892,175.022,16.757,152.567
C02346=1091.192,-27.228,-53.878,175.021,16.756,152.567
C02347=1091.186,-27.478,-53.866,175.019,16.754,152.567
C02348=1091.181,-27.727,-53.854,175.018,16.753,152.568
C02349=1091.175,-27.977,-53.841,175.016,16.752,152.567
C02350=1091.169,-28.227,-53.829,175.014,16.750,152.568
C02351=1091.162,-28.476,-53.816,175.012,16.749,152.568
C02352=1091.156,-28.726,-53.803,175.011,16.747,152.568
C02353=1091.150,-28.975,-53.791,175.009,16.746,152.568
C02354=1091.145,-29.225,-53.779,175.008,16.745,152.568
C02355=1091.139,-29.474,-53.766,175.006,16.744,152.568
C02356=1091.133,-29.724,-53.753,175.005,16.742,152.568
C02357=1091.127,-29.974,-53.740,175.002,16.741,152.568
C02358=1091.121,-30.224,-53.728,175.001,16.739,152.568
C02359=1091.116,-30.473,-53.715,174.999,16.738,152.568
C02360=1091.110,-30.723,-53.703,174.998,16.737,152.568
C02361=1091.104,-30.972,-53.690,174.996,16.736,152.568
C02362=1091.098,-31.222,-53.678,174.994,16.734,152.568
C02363=1091.091,-31.471,-53.665,174.993,16.733,152.569
C02364=1091.086,-31.720,-53.653,174.991,16.732,152.569
C02365=1091.080,-31.970,-53.640,174.989,16.730,152.569
C02366=1091.074,-32.220,-53.628,174.987,16.729,152.569
C02367=1091.068,-32.491,-53.614,174.986,16.727,152.569
C02368=1091.061,-32.761,-53.601,174.984,16.726,152.569
C02369=1091.055,-33.030,-53.588,174.982,16.724,152.569
C02370=1091.049,-33.300,-53.575,174.980,16.723,152.569
C02371=1091.043,-33.549,-53.562,174.979,16.722,152.569
C02372=1091.037,-33.799,-53.549,174.977,16.721,152.569
C02373=1091.031,-34.049,-53.536,174.976,16.719,152.569
C02374=1091.025,-34.298,-53.524,174.974,16.718,152.569
C02375=1091.019,-34.548,-53.512,174.973,16.717,152.569
C02376=1091.013,-34.798,-53.500,174.970,16.715,152.569
C02377=1091.008,-35.047,-53.488,174.969,16.714,152.570
C02378=1091.002,-35.297,-53.475,174.967,16.712,152.569
C02379=1090.996,-35.547,-53.462,174.966,16.711,152.570
C02380=1090.990,-35.797,-53.450,174.964,16.710,152.570
C02381=1090.984,-36.046,-53.438,174.963,16.708,152.570
C02382=1090.978,-36.295,-53.426,174.961,16.707,152.570
C02383=1090.972,-36.545,-53.413,174.960,16.706,152.570
C02384=1090.967,-36.794,-53.401,174.958,16.705,152.570
C02385=1090.961,-37.044,-53.388,174.956,16.703,152.570
C02386=1090.955,-37.295,-53.377,174.954,16.702,152.570
C02387=1090.950,-37.544,-53.364,174.953,16.701,152.570
C02388=1090.943,-37.794,-53.352,174.951,16.700,152.570
C02389=1090.937,-38.043,-53.340,174.950,16.698,152.570
C02390=1090.932,-38.293,-53.328,174.948,16.697,152.570
C02391=1090.926,-38.543,-53.315,174.946,16.696,152.570
C02392=1090.920,-38.792,-53.303,174.945,16.694,152.570
C02393=1090.914,-39.041,-53.291,174.943,16.693,152.570
C02394=1090.908,-39.291,-53.278,174.942,16.692,152.571
C02395=1090.902,-39.541,-53.266,174.940,16.691,152.571
C02396=1090.896,-39.790,-53.254,174.938,16.689,152.571
C02397=1090.891,-40.040,-53.242,174.936,16.687,152.571
C02398=1090.884,-40.290,-53.231,174.935,16.686,152.571
C02399=1090.878,-40.540,-53.218,174.933,16.685,152.571
C02400=1090.873,-40.789,-53.206,174.932,16.684,152.571
C02401=1090.866,-41.039,-53.194,174.930,16.683,152.571
C02402=1090.860,-41.289,-53.181,174.929,16.681,152.571
C02403=1090.855,-41.538,-53.169,174.927,16.680,152.571
C02404=1090.849,-41.788,-53.158,174.925,16.679,152.571
C02405=1090.843,-42.038,-53.145,174.924,16.678,152.571
C02406=1090.837,-42.287,-53.133,174.922,16.676,152.571
C02407=1090.831,-42.537,-53.121,174.921,16.675,152.572
C02408=1090.825,-42.786,-53.109,174.918,16.673,152.572
C02409=1090.819,-43.036,-53.098,174.917,16.672,152.572
C02410=1090.813,-43.286,-53.085,174.915,16.671,152.572
C02411=1090.808,-43.535,-53.073,174.914,16.670,152.572
C02412=1090.801,-43.785,-53.061,174.912,16.668,152.572
C02413=1090.795,-44.034,-53.048,174.911,16.667,152.572
C02414=1090.790,-44.284,-53.038,174.909,16.666,152.572
C02415=1090.784,-44.534,-53.025,174.907,16.665,152.572
C02416=1090.778,-44.784,-53.012,174.906,16.663,152.572
C02417=1090.772,-45.033,-53.001,174.904,16.662,152.572
C02418=1090.766,-45.283,-52.989,174.903,16.661,152.572
C02419=1090.760,-45.532,-52.977,174.901,16.660,152.572
C02420=1090.754,-45.782,-52.965,174.899,16.659,152.573
C02421=1090.748,-46.032,-52.954,174.898,16.657,152.573
C02422=1090.742,-46.281,-52.941,174.897,16.656,152.573
C02423=1090.737,-46.531,-52.929,174.894,16.655,152.573
C02424=1090.731,-46.780,-52.917,174.892,16.653,152.573
C02425=1090.725,-47.030,-52.905,174.891,16.652,152.573
C02426=1090.719,-47.279,-52.894,174.890,16.651,152.573
C02427=1090.713,-47.529,-52.881,174.888,16.650,152.573
C02428=1090.707,-47.779,-52.870,174.886,16.648,152.573
C02429=1090.701,-48.029,-52.858,174.885,16.647,152.573
C02430=1090.695,-48.279,-52.847,174.883,16.646,152.573
C02431=1090.689,-48.549,-52.833,174.882,16.645,152.573
C02432=1090.682,-48.820,-52.821,174.880,16.643,152.573
C02433=1090.676,-49.090,-52.808,174.878,16.642,152.574
C02434=1090.671,-49.360,-52.795,174.876,16.641,152.574
C02435=1090.664,-49.609,-52.783,174.875,16.639,152.574
C02436=1090.659,-49.859,-52.771,174.873,16.638,152.574
C02437=1090.652,-50.109,-52.760,174.871,16.637,152.574
C02438=1090.646,-50.359,-52.747,174.870,16.636,152.574
C02439=1090.641,-50.608,-52.736,174.868,16.634,152.574
C02440=1090.634,-50.858,-52.724,174.867,16.633,152.574
C02441=1090.629,-51.107,-52.712,174.865,16.632,152.574
C02442=1090.622,-51.357,-52.701,174.864,16.631,152.574
C02443=1090.616,-51.607,-52.689,174.862,16.629,152.574
C02444=1090.611,-51.857,-52.677,174.860,16.628,152.574
C02445=1090.604,-52.106,-52.665,174.859,16.627,152.575
C02446=1090.598,-52.356,-52.655,174.857,16.626,152.575
C02447=1090.592,-52.605,-52.642,174.856,16.625,152.575
C02448=1090.587,-52.855,-52.631,174.854,16.624,152.575
C02449=1090.580,-53.105,-52.619,174.852,16.623,152.575
C02450=1090.573,-53.354,-52.607,174.851,16.622,152.575
C02451=1090.568,-53.604,-52.596,174.849,16.621,152.575
C02452=1090.562,-53.853,-52.584,174.848,16.619,152.575
C02453=1090.556,-54.103,-52.573,174.846,16.618,152.575
C02454=1090.550,-54.353,-52.560,174.844,16.617,152.575
C02455=1090.544,-54.602,-52.550,174.843,16.616,152.575
C02456=1090.538,-54.852,-52.538,174.841,16.614,152.576
C02457=1090.531,-55.102,-52.526,174.840,16.613,152.576
C02458=1090.526,-55.352,-52.515,174.838,16.612,152.576
C02459=1090.520,-55.601,-52.503,174.836,16.611,152.576
C02460=1090.514,-55.851,-52.492,174.835,16.610,152.576
C02461=1090.507,-56.101,-52.480,174.833,16.609,152.576
C02462=1090.502,-56.350,-52.469,174.831,16.608,152.576
C02463=1090.496,-56.600,-52.457,174.830,16.607,152.576
C02464=1090.490,-56.849,-52.446,174.829,16.605,152.576
C02465=1090.483,-57.099,-52.434,174.827,16.604,152.576
C02466=1090.478,-57.348,-52.423,174.825,16.603,152.576
C02467=1090.472,-57.599,-52.411,174.824,16.602,152.577
C02468=1090.466,-57.848,-52.399,174.822,16.600,152.577
C02469=1090.460,-58.098,-52.388,174.820,16.599,152.577
C02470=1090.454,-58.347,-52.377,174.819,16.598,152.577
C02471=1090.448,-58.597,-52.365,174.817,16.597,152.577
C02472=1090.442,-58.847,-52.354,174.816,16.596,152.577
C02473=1090.436,-59.096,-52.342,174.814,16.595,152.577
C02474=1090.430,-59.346,-52.331,174.812,16.594,152.577
C02475=1090.423,-59.596,-52.320,174.811,16.593,152.577
C02476=1090.418,-59.845,-52.308,174.809,16.591,152.578
C02477=1090.412,-60.096,-52.296,174.808,16.590,152.577
C02478=1090.406,-60.345,-52.286,174.806,16.589,152.578
C02479=1090.400,-60.594,-52.274,174.804,16.588,152.578
C02480=1090.394,-60.844,-52.263,174.803,16.586,152.578
C02481=1090.389,-61.094,-52.251,174.801,16.585,152.578
C02482=1090.382,-61.343,-52.239,174.800,16.584,152.578
C02483=1090.376,-61.593,-52.228,174.798,16.583,152.578
C02484=1090.370,-61.843,-52.217,174.796,16.582,152.578
C02485=1090.364,-62.092,-52.206,174.795,16.581,152.578
C02486=1090.358,-62.342,-52.194,174.793,16.580,152.578
C02487=1090.353,-62.592,-52.183,174.791,16.579,152.579
C02488=1090.347,-62.841,-52.172,174.790,16.577,152.579
C02489=1090.340,-63.091,-52.160,174.788,16.576,152.579
C02490=1090.334,-63.341,-52.149,174.787,16.575,152.579
C02491=1090.328,-63.591,-52.138,174.785,16.574,152.579
C02492=1090.322,-63.840,-52.127,174.783,16.573,152.579
C02493=1090.317,-64.089,-52.115,174.782,16.572,152.579
C02494=1090.311,-64.340,-52.104,174.780,16.571,152.579
C02495=1090.304,-64.612,-52.092,174.779,16.569,152.579
C02496=1090.298,-64.883,-52.080,174.777,16.568,152.579
C02497=1090.291,-65.154,-52.067,174.776,16.567,152.579
C02498=1090.285,-65.426,-52.055,174.773,16.565,152.580
C02499=1090.279,-65.676,-52.044,174.772,16.564,152.580
C02500=1090.273,-65.925,-52.033,174.770,16.563,152.580
C02501=1090.267,-66.176,-52.022,174.769,16.562,152.580
C02502=1090.261,-66.424,-52.010,174.767,16.561,152.580
C02503=1090.255,-66.674,-51.999,174.766,16.560,152.580
C02504=1090.250,-66.924,-51.987,174.764,16.559,152.580
C02505=1090.244,-67.174,-51.977,174.763,16.558,152.580
C02506=1090.238,-67.423,-51.966,174.761,16.557,152.580
C02507=1090.232,-67.674,-51.954,174.759,16.556,152.581
C02508=1090.226,-67.923,-51.944,174.758,16.554,152.581
C02509=1090.220,-68.172,-51.932,174.756,16.553,152.581
C02510=1090.214,-68.422,-51.921,174.754,16.552,152.581
C02511=1090.208,-68.672,-51.910,174.753,16.551,152.581
C02512=1090.202,-68.921,-51.899,174.751,16.550,152.581
C02513=1090.196,-69.171,-51.888,174.750,16.549,152.581
C02514=1090.190,-69.421,-51.877,174.748,16.548,152.581
C02515=1090.185,-69.671,-51.865,174.746,16.547,152.581
C02516=1090.179,-69.921,-51.854,174.745,16.546,152.581
C02517=1090.173,-70.170,-51.843,174.743,16.544,152.582
C02518=1090.167,-70.420,-51.832,174.742,16.543,152.582
C02519=1090.161,-70.670,-51.821,174.740,16.542,152.582
C02520=1090.155,-70.919,-51.810,174.738,16.541,152.582
C02521=1090.149,-71.169,-51.799,174.737,16.540,152.582
C02522=1090.144,-71.418,-51.788,174.736,16.539,152.582
C02523=1090.137,-71.669,-51.777,174.734,16.538,152.582
C02524=1090.132,-71.918,-51.766,174.733,16.537,152.582
C02525=1090.126,-72.168,-51.755,174.731,16.536,152.582
C02526=1090.120,-72.417,-51.745,174.729,16.535,152.583
C02527=1090.114,-72.667,-51.733,174.728,16.534,152.583
C02528=1090.108,-72.917,-51.722,174.726,16.533,152.583
C02529=1090.102,-73.166,-51.712,174.724,16.531,152.583
C02530=1090.097,-73.416,-51.701,174.723,16.530,152.583
C02531=1090.090,-73.666,-51.689,174.721,16.529,152.583
C02532=1090.084,-73.915,-51.679,174.720,16.528,152.583
C02533=1090.079,-74.165,-51.668,174.718,16.527,152.583
C02534=1090.073,-74.414,-51.657,174.717,16.526,152.583
C02535=1090.067,-74.665,-51.646,174.716,16.525,152.583
C02536=1090.061,-74.914,-51.635,174.714,16.524,152.584
C02537=1090.055,-75.164,-51.624,174.712,16.523,152.584
C02538=1090.049,-75.414,-51.613,174.711,16.522,152.584
C02539=1090.043,-75.663,-51.602,174.709,16.521,152.584
C02540=1090.037,-75.912,-51.591,174.707,16.520,152.584
C02541=1090.030,-76.163,-51.580,174.706,16.519,152.584
C02542=1090.025,-76.412,-51.569,174.704,16.518,152.584
C02543=1090.019,-76.662,-51.558,174.702,16.517,152.584
C02544=1090.013,-76.911,-51.548,174.701,16.516,152.585
C02545=1090.007,-77.162,-51.537,174.700,16.515,152.585
C02546=1090.001,-77.411,-51.526,174.698,16.514,152.585
C02547=1089.995,-77.661,-51.516,174.697,16.513,152.585
C02548=1089.989,-77.910,-51.505,174.695,16.512,152.585
C02549=1089.983,-78.160,-51.494,174.693,16.511,152.585
C02550=1089.977,-78.410,-51.483,174.692,16.510,152.585
C02551=1089.971,-78.659,-51.472,174.690,16.509,152.585
C02552=1089.965,-78.909,-51.461,174.688,16.508,152.586
C02553=1089.959,-79.159,-51.451,174.687,16.507,152.586
C02554=1089.953,-79.409,-51.440,174.685,16.506,152.586
C02555=1089.947,-79.658,-51.429,174.684,16.505,152.586
C02556=1089.941,-79.908,-51.419,174.683,16.504,152.586
C02557=1089.934,-80.158,-51.408,174.681,16.503,152.586
C02558=1089.929,-80.407,-51.397,174.679,16.502,152.586
C02559=1089.923,-80.681,-51.386,174.677,16.501,152.586
C02560=1089.916,-80.955,-51.374,174.676,16.500,152.587
C02561=1089.909,-81.228,-51.363,174.674,16.499,152.587
C02562=1089.902,-81.503,-51.350,174.673,16.498,152.587
C02563=1089.896,-81.752,-51.340,174.671,16.497,152.587
C02564=1089.890,-82.002,-51.330,174.669,16.496,152.587
C02565=1089.884,-82.252,-51.319,174.667,16.495,152.587
C02566=1089.878,-82.502,-51.308,174.666,16.494,152.587
C02567=1089.872,-82.751,-51.298,174.664,16.493,152.588
C02568=1089.866,-83.001,-51.287,174.663,16.492,152.588
C02569=1089.860,-83.250,-51.277,174.661,16.491,152.588
C02570=1089.853,-83.500,-51.266,174.660,16.490,152.588
C02571=1089.848,-83.750,-51.255,174.658,16.489,152.588
C02572=1089.841,-84.000,-51.245,174.656,16.489,152.588
C02573=1089.836,-84.249,-51.235,174.655,16.487,152.588
C02574=1089.829,-84.498,-51.224,174.653,16.486,152.588
C02575=1089.823,-84.749,-51.214,174.652,16.486,152.589
C02576=1089.817,-84.999,-51.203,174.650,16.485,152.589
C02577=1089.811,-85.248,-51.193,174.649,16.484,152.589
C02578=1089.805,-85.497,-51.182,174.647,16.483,152.589
C02579=1089.799,-85.748,-51.171,174.645,16.482,152.589
C02580=1089.793,-85.997,-51.161,174.644,16.481,152.589
C02581=1089.787,-86.247,-51.150,174.642,16.480,152.589
C02582=1089.781,-86.497,-51.140,174.641,16.479,152.590
C02583=1089.775,-86.746,-51.130,174.639,16.478,152.590
C02584=1089.769,-86.995,-51.119,174.638,16.478,152.590
C02585=1089.762,-87.246,-51.109,174.636,16.477,152.590
C02586=1089.757,-87.496,-51.098,174.634,16.475,152.590
C02587=1089.750,-87.745,-51.088,174.633,16.474,152.590
C02588=1089.745,-87.995,-51.077,174.632,16.474,152.590
C02589=1089.738,-88.244,-51.067,174.630,16.473,152.591
C02590=1089.733,-88.494,-51.057,174.628,16.472,152.591
C02591=1089.726,-88.744,-51.046,174.627,16.471,152.591
C02592=1089.720,-88.994,-51.035,174.625,16.470,152.591
C02593=1089.715,-89.244,-51.025,174.623,16.469,152.591
C02594=1089.708,-89.493,-51.015,174.622,16.469,152.591
C02595=1089.703,-89.743,-51.005,174.620,16.468,152.591
C02596=1089.696,-89.992,-50.995,174.619,16.467,152.592
C02597=1089.691,-90.242,-50.984,174.617,16.466,152.592
C02598=1089.684,-90.492,-50.974,174.616,16.465,152.592
C02599=1089.678,-90.742,-50.963,174.614,16.464,152.592
C02600=1089.672,-90.991,-50.953,174.613,16.463,152.592
C02601=1089.666,-91.241,-50.942,174.611,16.462,152.592
C02602=1089.660,-91.491,-50.933,174.609,16.462,152.593
C02603=1089.654,-91.740,-50.922,174.608,16.461,152.593
C02604=1089.649,-91.990,-50.912,174.606,16.459,152.593
C02605=1089.642,-92.239,-50.902,174.604,16.459,152.593
C02606=1089.637,-92.490,-50.891,174.603,16.458,152.593
C02607=1089.630,-92.739,-50.881,174.602,16.457,152.593
C02608=1089.624,-92.990,-50.871,174.600,16.456,152.593
C02609=1089.618,-93.239,-50.860,174.598,16.455,152.594
C02610=1089.612,-93.489,-50.850,174.597,16.454,152.594
C02611=1089.606,-93.738,-50.840,174.596,16.454,152.594
C02612=1089.601,-93.988,-50.830,174.594,16.453,152.594
C02613=1089.594,-94.237,-50.819,174.592,16.452,152.594
C02614=1089.589,-94.487,-50.809,174.591,16.451,152.594
C02615=1089.582,-94.737,-50.799,174.589,16.450,152.594
C02616=1089.577,-94.987,-50.789,174.588,16.450,152.595
C02617=1089.571,-95.237,-50.779,174.586,16.449,152.595
C02618=1089.565,-95.486,-50.768,174.584,16.448,152.595
C02619=1089.559,-95.736,-50.759,174.583,16.447,152.595
C02620=1089.553,-95.985,-50.748,174.581,16.446,152.595
C02621=1089.547,-96.235,-50.738,174.580,16.446,152.595
C02622=1089.540,-96.485,-50.727,174.578,16.445,152.595
C02623=1089.534,-96.761,-50.717,174.577,16.443,152.596
C02624=1089.527,-97.037,-50.706,174.575,16.443,152.596
C02625=1089.520,-97.313,-50.695,174.573,16.442,152.596
C02626=1089.514,-97.589,-50.683,174.571,16.441,152.596
C02627=1089.508,-97.839,-50.673,174.570,16.440,152.596
C02628=1089.502,-98.089,-50.663,174.568,16.439,152.596
C02629=1089.496,-98.338,-50.653,174.567,16.439,152.597
C02630=1089.490,-98.589,-50.643,174.565,16.438,152.597
C02631=1089.484,-98.838,-50.633,174.563,16.437,152.597
C02632=1089.477,-99.087,-50.623,174.562,16.436,152.597
C02633=1089.472,-99.338,-50.613,174.560,16.435,152.597
C02634=1089.466,-99.587,-50.603,174.559,16.435,152.597
C02635=1089.459,-99.837,-50.593,174.557,16.434,152.598
C02636=1089.453,-100.087,-50.582,174.556,16.433,152.598
C02637=1089.447,-100.337,-50.572,174.554,16.432,152.598
C02638=1089.441,-100.586,-50.563,174.553,16.432,152.598
C02639=1089.434,-100.836,-50.553,174.551,16.431,152.598
C02640=1089.429,-101.086,-50.542,174.549,16.430,152.599
C02641=1089.423,-101.335,-50.533,174.548,16.429,152.599
C02642=1089.416,-101.585,-50.523,174.547,16.429,152.599
C02643=1089.411,-101.835,-50.513,174.545,16.428,152.599
C02644=1089.405,-102.085,-50.503,174.543,16.427,152.599
C02645=1089.398,-102.334,-50.493,174.541,16.426,152.599
C02646=1089.392,-102.584,-50.483,174.540,16.426,152.600
C02647=1089.386,-102.834,-50.473,174.539,16.425,152.600
C02648=1089.380,-103.083,-50.463,174.537,16.424,152.600
C02649=1089.374,-103.333,-50.453,174.535,16.423,152.600
C02650=1089.368,-103.583,-50.444,174.534,16.423,152.600
C02651=1089.362,-103.833,-50.433,174.532,16.422,152.600
C02652=1089.356,-104.082,-50.423,174.531,16.421,152.601
C02653=1089.350,-104.332,-50.414,174.529,16.420,152.601
C02654=1089.344,-104.582,-50.404,174.528,16.420,152.601
C02655=1089.337,-104.832,-50.395,174.526,16.419,152.601
C02656=1089.332,-105.081,-50.384,174.524,16.419,152.601
C02657=1089.326,-105.331,-50.374,174.523,16.417,152.601
C02658=1089.319,-105.581,-50.365,174.522,16.417,152.602
C02659=1089.313,-105.831,-50.355,174.520,16.416,152.602
C02660=1089.308,-106.081,-50.345,174.518,16.416,152.602
C02661=1089.301,-106.330,-50.335,174.516,16.415,152.602
C02662=1089.295,-106.580,-50.325,174.515,16.414,152.602
C02663=1089.289,-106.829,-50.316,174.513,16.414,152.603
C02664=1089.283,-107.079,-50.306,174.512,16.413,152.603
C02665=1089.277,-107.329,-50.296,174.510,16.412,152.603
C02666=1089.271,-107.579,-50.286,174.509,16.412,152.603
C02667=1089.265,-107.828,-50.276,174.507,16.411,152.603
C02668=1089.259,-108.078,-50.266,174.506,16.410,152.603
C02669=1089.252,-108.328,-50.257,174.504,16.410,152.604
C02670=1089.246,-108.578,-50.247,174.503,16.409,152.604
C02671=1089.240,-108.828,-50.238,174.501,16.408,152.604
C02672=1089.234,-109.077,-50.228,174.499,16.407,152.604
C02673=1089.228,-109.326,-50.219,174.498,16.407,152.604
C02674=1089.222,-109.576,-50.209,174.496,16.406,152.605
C02675=1089.216,-109.826,-50.199,174.494,16.406,152.605
C02676=1089.210,-110.076,-50.189,174.494,16.405,152.605
C02677=1089.204,-110.325,-50.179,174.492,16.405,152.605
C02678=1089.198,-110.575,-50.170,174.490,16.403,152.605
C02679=1089.192,-110.825,-50.160,174.488,16.403,152.606
C02680=1089.186,-111.075,-50.151,174.487,16.403,152.606
C02681=1089.179,-111.325,-50.141,174.485,16.402,152.606
C02682=1089.173,-111.574,-50.132,174.483,16.401,152.606
C02683=1089.167,-111.824,-50.122,174.482,16.401,152.606
C02684=1089.161,-112.074,-50.112,174.481,16.400,152.607
C02685=1089.155,-112.324,-50.103,174.479,16.399,152.607
C02686=1089.148,-112.574,-50.093,174.478,16.399,152.607
C02687=1089.142,-112.844,-50.083,174.476,16.398,152.607
C02688=1089.136,-113.113,-50.073,174.474,16.397,152.607
C02689=1089.129,-113.383,-50.062,174.472,16.397,152.608
C02690=1089.122,-113.652,-50.052,174.471,16.396,152.608
C02691=1089.116,-113.902,-50.042,174.470,16.396,152.608
C02692=1089.110,-114.152,-50.032,174.468,16.395,152.608
C02693=1089.104,-114.402,-50.023,174.466,16.394,152.608
C02694=1089.097,-114.652,-50.013,174.464,16.393,152.609
C02695=1089.091,-114.901,-50.004,174.463,16.393,152.609
C02696=1089.085,-115.152,-49.995,174.461,16.393,152.609
C02697=1089.079,-115.402,-49.985,174.459,16.392,152.609
C02698=1089.074,-115.651,-49.976,174.458,16.392,152.609
C02699=1089.067,-115.901,-49.967,174.456,16.391,152.610
C02700=1089.061,-116.150,-49.957,174.455,16.390,152.610
C02701=1089.055,-116.400,-49.947,174.454,16.390,152.610
C02702=1089.049,-116.650,-49.938,174.452,16.389,152.610
C02703=1089.043,-116.900,-49.928,174.450,16.389,152.611
C02704=1089.037,-117.149,-49.919,174.449,16.388,152.611
C02705=1089.030,-117.399,-49.909,174.447,16.387,152.611
C02706=1089.024,-117.649,-49.900,174.445,16.387,152.611
C02707=1089.018,-117.899,-49.890,174.444,16.387,152.611
C02708=1089.013,-118.148,-49.881,174.443,16.386,152.612
C02709=1089.006,-118.398,-49.871,174.441,16.385,152.612
C02710=1088.999,-118.647,-49.862,174.440,16.385,152.612
C02711=1088.994,-118.898,-49.853,174.438,16.384,152.612
C02712=1088.987,-119.147,-49.844,174.436,16.383,152.612
C02713=1088.981,-119.397,-49.834,174.435,16.383,152.613
C02714=1088.975,-119.647,-49.825,174.433,16.383,152.613
C02715=1088.969,-119.897,-49.815,174.431,16.382,152.613
C02716=1088.963,-120.146,-49.806,174.430,16.381,152.613
C02717=1088.957,-120.396,-49.796,174.428,16.381,152.614
C02718=1088.951,-120.646,-49.787,174.426,16.380,152.614
C02719=1088.944,-120.896,-49.779,174.425,16.380,152.614
C02720=1088.938,-121.145,-49.769,174.423,16.380,152.614
C02721=1088.932,-121.395,-49.759,174.423,16.379,152.614
C02722=1088.926,-121.644,-49.750,174.421,16.378,152.615
C02723=1088.920,-121.894,-49.741,174.419,16.378,152.615
C02724=1088.914,-122.144,-49.731,174.418,16.378,152.615
C02725=1088.908,-122.394,-49.722,174.416,16.377,152.615
C02726=1088.901,-122.644,-49.713,174.414,16.376,152.616
C02727=1088.895,-122.894,-49.704,174.413,16.376,152.616
C02728=1088.890,-123.143,-49.694,174.411,16.375,152.616
C02729=1088.884,-123.393,-49.686,174.409,16.375,152.616
C02730=1088.878,-123.643,-49.676,174.408,16.375,152.616
C02731=1088.871,-123.893,-49.666,174.406,16.374,152.617
C02732=1088.865,-124.142,-49.658,174.404,16.373,152.617
C02733=1088.858,-124.392,-49.648,174.403,16.373,152.617
C02734=1088.853,-124.642,-49.639,174.402,16.372,152.617
C02735=1088.847,-124.892,-49.630,174.400,16.372,152.618
C02736=1088.840,-125.141,-49.621,174.398,16.372,152.618
C02737=1088.834,-125.391,-49.611,174.397,16.371,152.618
C02738=1088.828,-125.641,-49.603,174.395,16.371,152.618
C02739=1088.822,-125.891,-49.593,174.394,16.370,152.619
C02740=1088.815,-126.140,-49.584,174.392,16.370,152.619
C02741=1088.809,-126.390,-49.575,174.391,16.370,152.619
C02742=1088.803,-126.640,-49.566,174.389,16.369,152.619
C02743=1088.797,-126.890,-49.556,174.388,16.369,152.619
C02744=1088.790,-127.139,-49.547,174.386,16.368,152.620
C02745=1088.785,-127.389,-49.539,174.384,16.367,152.620
C02746=1088.779,-127.639,-49.529,174.383,16.367,152.620
C02747=1088.772,-127.897,-49.520,174.381,16.367,152.620
C02748=1088.766,-128.155,-49.511,174.380,16.367,152.621
C02749=1088.766,-128.413,-49.499,174.379,16.365,152.620
C02750=1088.773,-128.668,-49.486,174.378,16.360,152.620
C02751=1088.368,-128.689,-49.610,174.337,16.466,152.648
C02752=1088.362,-128.435,-49.623,174.337,16.470,152.649
C02753=1088.362,-128.177,-49.635,174.338,16.472,152.649
C02754=1088.367,-127.919,-49.644,174.340,16.472,152.649
C02755=1088.373,-127.661,-49.654,174.341,16.472,152.648
C02756=1088.380,-127.411,-49.663,174.343,16.473,152.648
C02757=1088.386,-127.161,-49.672,174.344,16.474,152.648
C02758=1088.392,-126.912,-49.681,174.346,16.474,152.648
C02759=1088.398,-126.662,-49.690,174.348,16.475,152.648
C02760=1088.404,-126.412,-49.699,174.349,16.475,152.647
C02761=1088.411,-126.162,-49.708,174.351,16.475,152.647
C02762=1088.417,-125.912,-49.718,174.353,16.476,152.647
C02763=1088.423,-125.662,-49.727,174.354,16.476,152.647
C02764=1088.429,-125.413,-49.735,174.356,16.477,152.646
C02765=1088.435,-125.163,-49.745,174.357,16.477,152.646
C02766=1088.441,-124.913,-49.754,174.358,16.478,152.646
C02767=1088.448,-124.664,-49.763,174.360,16.478,152.646
C02768=1088.454,-124.414,-49.772,174.361,16.478,152.646
C02769=1088.460,-124.164,-49.781,174.363,16.479,152.645
C02770=1088.466,-123.915,-49.791,174.365,16.480,152.645
C02771=1088.472,-123.665,-49.801,174.366,16.480,152.645
C02772=1088.478,-123.414,-49.809,174.368,16.481,152.645
C02773=1088.485,-123.165,-49.818,174.370,16.481,152.644
C02774=1088.491,-122.915,-49.828,174.371,16.481,152.644
C02775=1088.496,-122.666,-49.837,174.373,16.482,152.644
C02776=1088.503,-122.416,-49.847,174.375,16.483,152.644
C02777=1088.508,-122.166,-49.856,174.376,16.483,152.644
C02778=1088.515,-121.916,-49.865,174.378,16.484,152.643
C02779=1088.522,-121.667,-49.874,174.379,16.484,152.643
C02780=1088.528,-121.417,-49.884,174.380,16.485,152.643
C02781=1088.533,-121.168,-49.893,174.382,16.486,152.643
C02782=1088.539,-120.918,-49.902,174.383,16.486,152.643
C02783=1088.545,-120.667,-49.911,174.385,16.486,152.642
C02784=1088.552,-120.418,-49.921,174.387,16.487,152.642
C02785=1088.558,-120.168,-49.930,174.388,16.487,152.642
C02786=1088.565,-119.918,-49.939,174.390,16.488,152.642
C02787=1088.571,-119.669,-49.949,174.392,16.489,152.641
C02788=1088.576,-119.420,-49.958,174.393,16.489,152.641
C02789=1088.583,-119.170,-49.968,174.395,16.490,152.641
C02790=1088.588,-118.919,-49.977,174.396,16.490,152.641
C02791=1088.595,-118.670,-49.986,174.398,16.490,152.641
C02792=1088.601,-118.420,-49.996,174.399,16.491,152.640
C02793=1088.607,-118.170,-50.005,174.401,16.492,152.640
C02794=1088.613,-117.920,-50.015,174.402,16.492,152.640
C02795=1088.619,-117.670,-50.024,174.404,16.493,152.640
C02796=1088.626,-117.422,-50.033,174.406,16.494,152.640
C02797=1088.632,-117.172,-50.043,174.407,16.494,152.639
C02798=1088.638,-116.922,-50.052,174.409,16.494,152.639
C02799=1088.644,-116.672,-50.062,174.410,16.496,152.639
C02800=1088.650,-116.422,-50.071,174.412,16.496,152.639
C02801=1088.656,-116.173,-50.081,174.413,16.496,152.639
C02802=1088.663,-115.923,-50.090,174.415,16.497,152.638
C02803=1088.668,-115.672,-50.099,174.417,16.498,152.638
C02804=1088.675,-115.423,-50.109,174.418,16.498,152.638
C02805=1088.681,-115.173,-50.118,174.420,16.499,152.638
C02806=1088.686,-114.924,-50.128,174.422,16.500,152.638
C02807=1088.693,-114.674,-50.137,174.423,16.500,152.637
C02808=1088.699,-114.424,-50.147,174.424,16.501,152.637
C02809=1088.705,-114.174,-50.156,174.426,16.501,152.637
C02810=1088.711,-113.924,-50.166,174.427,16.501,152.637
C02811=1088.717,-113.675,-50.175,174.429,16.503,152.637
C02812=1088.723,-113.404,-50.186,174.431,16.503,152.636
C02813=1088.731,-113.135,-50.196,174.433,16.504,152.636
C02814=1088.737,-112.864,-50.207,174.434,16.505,152.636
C02815=1088.743,-112.594,-50.217,174.436,16.505,152.636
C02816=1088.749,-112.344,-50.227,174.437,16.506,152.636
C02817=1088.755,-112.094,-50.237,174.439,16.507,152.635
C02818=1088.762,-111.845,-50.246,174.441,16.507,152.635
C02819=1088.768,-111.595,-50.256,174.442,16.508,152.635
C02820=1088.774,-111.345,-50.265,174.444,16.508,152.635
C02821=1088.780,-111.095,-50.275,174.445,16.510,152.635
C02822=1088.786,-110.846,-50.284,174.446,16.510,152.634
C02823=1088.792,-110.596,-50.294,174.448,16.510,152.634
C02824=1088.799,-110.346,-50.304,174.450,16.511,152.634
C02825=1088.805,-110.096,-50.313,174.452,16.512,152.634
C02826=1088.811,-109.847,-50.323,174.453,16.512,152.634
C02827=1088.817,-109.597,-50.333,174.455,16.513,152.633
C02828=1088.824,-109.347,-50.343,174.457,16.514,152.633
C02829=1088.830,-109.098,-50.352,174.457,16.514,152.633
C02830=1088.835,-108.847,-50.362,174.459,16.515,152.633
C02831=1088.841,-108.598,-50.372,174.461,16.516,152.633
C02832=1088.848,-108.348,-50.381,174.463,16.517,152.632
C02833=1088.854,-108.098,-50.391,174.464,16.517,152.632
C02834=1088.860,-107.850,-50.401,174.466,16.518,152.632
C02835=1088.866,-107.600,-50.410,174.467,16.519,152.632
C02836=1088.872,-107.350,-50.420,174.468,16.519,152.632
C02837=1088.878,-107.100,-50.430,174.470,16.520,152.632
C02838=1088.884,-106.850,-50.440,174.472,16.521,152.631
C02839=1088.890,-106.600,-50.449,174.473,16.522,152.631
C02840=1088.896,-106.350,-50.459,174.475,16.522,152.631
C02841=1088.902,-106.101,-50.469,174.476,16.523,152.631
C02842=1088.909,-105.851,-50.479,174.478,16.523,152.631
C02843=1088.914,-105.601,-50.489,174.480,16.525,152.631
C02844=1088.920,-105.352,-50.498,174.481,16.525,152.630
C02845=1088.926,-105.102,-50.508,174.482,16.526,152.630
C02846=1088.933,-104.853,-50.518,174.484,16.526,152.630
C02847=1088.939,-104.603,-50.528,174.486,16.527,152.630
C02848=1088.944,-104.353,-50.538,174.487,16.528,152.630
C02849=1088.951,-104.103,-50.548,174.489,16.529,152.630
C02850=1088.957,-103.854,-50.558,174.491,16.529,152.629
C02851=1088.963,-103.604,-50.567,174.492,16.530,152.629
C02852=1088.969,-103.354,-50.578,174.493,16.530,152.629
C02853=1088.975,-103.104,-50.587,174.495,16.532,152.629
C02854=1088.981,-102.855,-50.597,174.497,16.533,152.629
C02855=1088.988,-102.605,-50.607,174.499,16.533,152.629
C02856=1088.993,-102.355,-50.617,174.499,16.534,152.628
C02857=1088.999,-102.105,-50.627,174.501,16.534,152.628
C02858=1089.006,-101.856,-50.637,174.503,16.536,152.628
C02859=1089.011,-101.606,-50.647,174.505,16.536,152.628
C02860=1089.017,-101.356,-50.657,174.506,16.537,152.628
C02861=1089.023,-101.106,-50.666,174.507,16.538,152.628
C02862=1089.030,-100.857,-50.677,174.509,16.538,152.627
C02863=1089.035,-100.607,-50.687,174.511,16.540,152.627
C02864=1089.041,-100.357,-50.696,174.513,16.540,152.627
C02865=1089.049,-100.107,-50.707,174.513,16.541,152.627
C02866=1089.055,-99.857,-50.717,174.515,16.541,152.627
C02867=1089.060,-99.607,-50.727,174.517,16.542,152.627
C02868=1089.067,-99.358,-50.737,174.519,16.544,152.626
C02869=1089.073,-99.108,-50.747,174.520,16.544,152.626
C02870=1089.078,-98.858,-50.757,174.521,16.545,152.626
C02871=1089.085,-98.609,-50.767,174.523,16.545,152.626
C02872=1089.091,-98.359,-50.777,174.525,16.546,152.626
C02873=1089.097,-98.110,-50.787,174.527,16.548,152.626
C02874=1089.103,-97.860,-50.797,174.528,16.548,152.625
C02875=1089.109,-97.610,-50.807,174.529,16.549,152.625
C02876=1089.116,-97.334,-50.818,174.531,16.550,152.625
C02877=1089.123,-97.058,-50.830,174.533,16.550,152.625
C02878=1089.129,-96.781,-50.840,174.534,16.552,152.625
C02879=1089.136,-96.505,-50.852,174.536,16.553,152.625
C02880=1089.141,-96.256,-50.862,174.538,16.553,152.624
C02881=1089.148,-96.006,-50.872,174.540,16.554,152.624
C02882=1089.153,-95.756,-50.882,174.541,16.555,152.624
C02883=1089.159,-95.507,-50.892,174.542,16.556,152.624
C02884=1089.165,-95.256,-50.903,174.544,16.557,152.624
C02885=1089.171,-95.007,-50.913,174.546,16.558,152.624
C02886=1089.177,-94.757,-50.923,174.547,16.559,152.624
C02887=1089.183,-94.508,-50.933,174.549,16.559,152.623
C02888=1089.189,-94.258,-50.944,174.550,16.560,152.623
C02889=1089.196,-94.008,-50.954,174.552,16.561,152.623
C02890=1089.201,-93.758,-50.964,174.553,16.562,152.623
C02891=1089.207,-93.508,-50.974,174.555,16.563,152.623
C02892=1089.213,-93.259,-50.985,174.557,16.564,152.623
C02893=1089.219,-93.009,-50.994,174.558,16.565,152.623
C02894=1089.225,-92.759,-51.005,174.559,16.565,152.622
C02895=1089.231,-92.510,-51.015,174.561,16.566,152.622
C02896=1089.237,-92.260,-51.026,174.563,16.567,152.622
C02897=1089.243,-92.010,-51.035,174.564,16.568,152.622
C02898=1089.249,-91.761,-51.046,174.566,16.569,152.622
C02899=1089.255,-91.512,-51.056,174.567,16.570,152.622
C02900=1089.261,-91.261,-51.067,174.569,16.571,152.622
C02901=1089.267,-91.011,-51.078,174.570,16.572,152.622
C02902=1089.273,-90.761,-51.087,174.572,16.572,152.621
C02903=1089.279,-90.512,-51.098,174.574,16.574,152.621
C02904=1089.285,-90.262,-51.108,174.575,16.575,152.621
C02905=1089.291,-90.013,-51.119,174.576,16.575,152.621
C02906=1089.297,-89.763,-51.128,174.578,16.576,152.621
C02907=1089.303,-89.513,-51.139,174.580,16.577,152.621
C02908=1089.310,-89.264,-51.150,174.581,16.578,152.621
C02909=1089.315,-89.013,-51.160,174.583,16.579,152.620
C02910=1089.322,-88.764,-51.170,174.585,16.580,152.620
C02911=1089.327,-88.514,-51.180,174.586,16.580,152.620
C02912=1089.333,-88.265,-51.191,174.587,16.582,152.620
C02913=1089.339,-88.015,-51.202,174.589,16.583,152.620
C02914=1089.345,-87.765,-51.212,174.591,16.584,152.620
C02915=1089.352,-87.515,-51.222,174.593,16.584,152.619
C02916=1089.358,-87.266,-51.233,174.594,16.585,152.619
C02917=1089.364,-87.016,-51.243,174.595,16.586,152.619
C02918=1089.370,-86.767,-51.254,174.597,16.587,152.619
C02919=1089.375,-86.517,-51.264,174.598,16.588,152.619
C02920=1089.382,-86.267,-51.275,174.600,16.589,152.619
C02921=1089.388,-86.017,-51.285,174.602,16.590,152.619
C02922=1089.394,-85.767,-51.295,174.603,16.591,152.619
C02923=1089.400,-85.518,-51.306,174.605,16.592,152.619
C02924=1089.406,-85.268,-51.317,174.606,16.593,152.618
C02925=1089.413,-85.019,-51.327,174.608,16.593,152.618
C02926=1089.418,-84.768,-51.338,174.609,16.595,152.618
C02927=1089.425,-84.519,-51.348,174.611,16.596,152.618
C02928=1089.430,-84.270,-51.359,174.613,16.597,152.618
C02929=1089.436,-84.020,-51.369,174.614,16.598,152.618
C02930=1089.443,-83.770,-51.379,174.616,16.599,152.618
C02931=1089.449,-83.520,-51.390,174.618,16.600,152.617
C02932=1089.454,-83.271,-51.401,174.619,16.600,152.617
C02933=1089.460,-83.021,-51.411,174.620,16.601,152.617
C02934=1089.467,-82.771,-51.422,174.622,16.602,152.617
C02935=1089.473,-82.522,-51.432,174.623,16.603,152.617
C02936=1089.479,-82.272,-51.443,174.625,16.604,152.617
C02937=1089.484,-82.022,-51.453,174.627,16.605,152.617
C02938=1089.491,-81.772,-51.464,174.629,16.606,152.617
C02939=1089.497,-81.523,-51.475,174.629,16.607,152.616
C02940=1089.504,-81.249,-51.486,174.632,16.609,152.616
C02941=1089.511,-80.974,-51.498,174.634,16.610,152.616
C02942=1089.518,-80.701,-51.509,174.635,16.610,152.616
C02943=1089.524,-80.427,-51.522,174.637,16.611,152.616
C02944=1089.530,-80.177,-51.532,174.639,16.613,152.616
C02945=1089.537,-79.928,-51.543,174.640,16.614,152.616
C02946=1089.542,-79.677,-51.553,174.641,16.614,152.616
C02947=1089.548,-79.428,-51.564,174.643,16.615,152.615
C02948=1089.554,-79.178,-51.575,174.644,16.616,152.615
C02949=1089.560,-78.928,-51.586,174.646,16.618,152.615
C02950=1089.566,-78.679,-51.597,174.648,16.619,152.615
C02951=1089.572,-78.430,-51.607,174.649,16.620,152.615
C02952=1089.578,-78.179,-51.618,174.651,16.621,152.615
C02953=1089.584,-77.929,-51.629,174.652,16.622,152.615
C02954=1089.590,-77.680,-51.640,174.654,16.623,152.615
C02955=1089.595,-77.430,-51.651,174.655,16.623,152.614
C02956=1089.602,-77.181,-51.661,174.657,16.624,152.614
C02957=1089.608,-76.931,-51.672,174.658,16.625,152.614
C02958=1089.614,-76.681,-51.683,174.660,16.627,152.614
C02959=1089.620,-76.432,-51.694,174.662,16.628,152.614
C02960=1089.625,-76.182,-51.705,174.663,16.629,152.614
C02961=1089.632,-75.932,-51.715,174.665,16.630,152.614
C02962=1089.638,-75.682,-51.726,174.667,16.631,152.614
C02963=1089.644,-75.433,-51.736,174.668,16.632,152.614
C02964=1089.650,-75.183,-51.748,174.670,16.633,152.613
C02965=1089.656,-74.933,-51.759,174.671,16.634,152.613
C02966=1089.662,-74.684,-51.769,174.673,16.635,152.613
C02967=1089.667,-74.434,-51.780,174.674,16.636,152.613
C02968=1089.674,-74.184,-51.792,174.676,16.637,152.613
C02969=1089.679,-73.935,-51.802,174.677,16.638,152.613
C02970=1089.685,-73.685,-51.813,174.679,16.639,152.613
C02971=1089.691,-73.435,-51.825,174.680,16.640,152.613
C02972=1089.697,-73.185,-51.835,174.682,16.642,152.613
C02973=1089.703,-72.936,-51.846,174.684,16.643,152.613
C02974=1089.709,-72.687,-51.857,174.685,16.644,152.612
C02975=1089.715,-72.436,-51.868,174.687,16.645,152.612
C02976=1089.721,-72.187,-51.879,174.689,16.646,152.612
C02977=1089.726,-71.937,-51.890,174.690,16.647,152.612
C02978=1089.732,-71.688,-51.901,174.692,16.648,152.612
C02979=1089.739,-71.438,-51.912,174.693,16.649,152.612
C02980=1089.744,-71.188,-51.923,174.695,16.651,152.612
C02981=1089.750,-70.939,-51.934,174.696,16.652,152.612
C02982=1089.756,-70.689,-51.945,174.697,16.653,152.612
C02983=1089.762,-70.439,-51.956,174.699,16.654,152.612
C02984=1089.768,-70.190,-51.967,174.700,16.655,152.612
C02985=1089.774,-69.940,-51.978,174.702,16.656,152.611
C02986=1089.779,-69.690,-51.990,174.704,16.657,152.611
C02987=1089.785,-69.440,-52.001,174.705,16.658,152.611
C02988=1089.791,-69.191,-52.012,174.707,16.659,152.611
C02989=1089.797,-68.941,-52.023,174.709,16.661,152.611
C02990=1089.803,-68.691,-52.034,174.710,16.662,152.611
C02991=1089.809,-68.442,-52.045,174.712,16.663,152.611
C02992=1089.815,-68.192,-52.056,174.713,16.664,152.611
C02993=1089.821,-67.942,-52.067,174.715,16.666,152.611
C02994=1089.827,-67.693,-52.078,174.716,16.667,152.611
C02995=1089.833,-67.443,-52.089,174.718,16.668,152.611
C02996=1089.839,-67.193,-52.100,174.720,16.669,152.610
C02997=1089.844,-66.944,-52.113,174.721,16.670,152.610
C02998=1089.850,-66.694,-52.124,174.723,16.671,152.610
C02999=1089.856,-66.444,-52.135,174.725,16.672,152.610
C03000=1089.862,-66.195,-52.146,174.726,16.673,152.610
C03001=1089.868,-65.945,-52.157,174.728,16.674,152.610
C03002=1089.874,-65.695,-52.168,174.729,16.676,152.610
C03003=1089.880,-65.446,-52.179,174.731,16.677,152.610
C03004=1089.886,-65.174,-52.192,174.732,16.678,152.610
C03005=1089.893,-64.902,-52.204,174.734,16.679,152.610
C03006=1089.899,-64.630,-52.216,174.736,16.681,152.610
C03007=1089.905,-64.358,-52.228,174.737,16.682,152.609
C03008=1089.912,-64.109,-52.240,174.739,16.683,152.609
C03009=1089.917,-63.859,-52.251,174.740,16.684,152.609
C03010=1089.924,-63.609,-52.262,174.742,16.685,152.609
C03011=1089.929,-63.360,-52.273,174.744,16.686,152.609
C03012=1089.936,-63.110,-52.285,174.745,16.688,152.609
C03013=1089.941,-62.860,-52.296,174.747,16.689,152.609
C03014=1089.947,-62.611,-52.307,174.748,16.690,152.609
C03015=1089.953,-62.361,-52.318,174.750,16.691,152.609
C03016=1089.959,-62.112,-52.330,174.752,16.692,152.609
C03017=1089.965,-61.862,-52.341,174.753,16.693,152.608
C03018=1089.971,-61.612,-52.352,174.755,16.694,152.608
C03019=1089.977,-61.362,-52.365,174.756,16.696,152.608
C03020=1089.983,-61.113,-52.376,174.758,16.697,152.608
C03021=1089.989,-60.863,-52.387,174.759,16.698,152.608
C03022=1089.995,-60.613,-52.398,174.761,16.699,152.608
C03023=1090.001,-60.364,-52.409,174.763,16.701,152.608
C03024=1090.007,-60.114,-52.421,174.764,16.702,152.608
C03025=1090.012,-59.864,-52.432,174.766,16.703,152.608
C03026=1090.019,-59.615,-52.444,174.768,16.704,152.608
C03027=1090.025,-59.365,-52.455,174.769,16.705,152.608
C03028=1090.031,-59.115,-52.466,174.770,16.707,152.608
C03029=1090.036,-58.866,-52.478,174.772,16.708,152.608
C03030=1090.043,-58.616,-52.490,174.774,16.709,152.607
C03031=1090.049,-58.367,-52.501,174.775,16.710,152.607
C03032=1090.055,-58.117,-52.512,174.777,16.711,152.607
C03033=1090.061,-57.867,-52.523,174.779,16.712,152.607
C03034=1090.067,-57.617,-52.536,174.780,16.713,152.607
C03035=1090.072,-57.368,-52.547,174.782,16.715,152.607
C03036=1090.079,-57.118,-52.559,174.783,16.716,152.607
C03037=1090.085,-56.869,-52.570,174.785,16.717,152.607
C03038=1090.090,-56.618,-52.581,174.786,16.718,152.607
C03039=1090.097,-56.369,-52.593,174.788,16.719,152.607
C03040=1090.103,-56.119,-52.604,174.790,16.721,152.606
C03041=1090.109,-55.870,-52.616,174.791,16.722,152.606
C03042=1090.114,-55.620,-52.628,174.793,16.723,152.606
C03043=1090.121,-55.371,-52.639,174.794,16.724,152.606
C03044=1090.127,-55.121,-52.650,174.796,16.726,152.606
C03045=1090.133,-54.872,-52.662,174.798,16.727,152.606
C03046=1090.139,-54.621,-52.674,174.799,16.728,152.606
C03047=1090.145,-54.372,-52.686,174.801,16.729,152.606
C03048=1090.151,-54.122,-52.697,174.802,16.730,152.606
C03049=1090.158,-53.873,-52.709,174.804,16.732,152.606
C03050=1090.163,-53.623,-52.720,174.805,16.733,152.606
C03051=1090.169,-53.373,-52.732,174.807,16.734,152.606
C03052=1090.175,-53.124,-52.743,174.809,16.735,152.606
C03053=1090.182,-52.874,-52.755,174.810,16.736,152.605
C03054=1090.187,-52.624,-52.767,174.812,16.737,152.605
C03055=1090.193,-52.375,-52.778,174.814,16.738,152.605
C03056=1090.200,-52.125,-52.790,174.815,16.740,152.605
C03057=1090.205,-51.875,-52.802,174.816,16.741,152.605
C03058=1090.211,-51.625,-52.813,174.818,16.742,152.605
C03059=1090.218,-51.376,-52.825,174.820,16.743,152.605
C03060=1090.223,-51.126,-52.837,174.821,16.744,152.605
C03061=1090.230,-50.876,-52.848,174.823,16.745,152.605
C03062=1090.236,-50.627,-52.860,174.824,16.747,152.605
C03063=1090.241,-50.377,-52.872,174.827,16.749,152.605
C03064=1090.247,-50.128,-52.883,174.828,16.750,152.605
C03065=1090.253,-49.878,-52.896,174.830,16.751,152.604
C03066=1090.259,-49.628,-52.907,174.831,16.753,152.604
C03067=1090.265,-49.379,-52.919,174.833,16.754,152.604
C03068=1090.271,-49.108,-52.932,174.835,16.755,152.604
C03069=1090.278,-48.838,-52.945,174.836,16.756,152.604
C03070=1090.284,-48.567,-52.958,174.838,16.758,152.604
C03071=1090.290,-48.297,-52.970,174.840,16.759,152.604
C03072=1090.296,-48.047,-52.983,174.842,16.760,152.604
C03073=1090.302,-47.798,-52.994,174.843,16.762,152.604
C03074=1090.308,-47.547,-53.006,174.845,16.763,152.604
C03075=1090.314,-47.299,-53.018,174.846,16.764,152.604
C03076=1090.320,-47.049,-53.030,174.848,16.765,152.604
C03077=1090.326,-46.798,-53.041,174.849,16.767,152.604
C03078=1090.331,-46.549,-53.054,174.851,16.768,152.604
C03079=1090.337,-46.299,-53.066,174.852,16.769,152.604
C03080=1090.343,-46.050,-53.077,174.854,16.771,152.604
C03081=1090.349,-45.800,-53.090,174.855,16.772,152.603
C03082=1090.356,-45.550,-53.102,174.857,16.773,152.603
C03083=1090.361,-45.301,-53.114,174.859,16.774,152.603
C03084=1090.367,-45.051,-53.125,174.860,16.776,152.603
C03085=1090.372,-44.802,-53.137,174.862,16.778,152.603
C03086=1090.378,-44.552,-53.150,174.864,16.779,152.603
C03087=1090.385,-44.302,-53.162,174.866,16.780,152.603
C03088=1090.390,-44.053,-53.173,174.867,16.781,152.603
C03089=1090.397,-43.803,-53.185,174.869,16.782,152.603
C03090=1090.403,-43.553,-53.198,174.870,16.784,152.603
C03091=1090.408,-43.304,-53.210,174.872,16.785,152.603
C03092=1090.414,-43.054,-53.221,174.873,16.786,152.603
C03093=1090.420,-42.805,-53.233,174.875,16.787,152.603
C03094=1090.426,-42.555,-53.245,174.877,16.789,152.603
C03095=1090.432,-42.305,-53.258,174.878,16.790,152.603
C03096=1090.438,-42.066,-53.269,174.879,16.791,152.602
C03097=1090.443,-41.826,-53.281,174.881,16.792,152.602
C03098=1090.449,-41.586,-53.293,174.883,16.794,152.602
C03099=1090.454,-41.346,-53.304,174.884,16.795,152.602
C03100=1090.460,-41.107,-53.316,174.886,16.796,152.602
C03101=1090.467,-40.867,-53.328,174.887,16.797,152.602
C03102=1090.472,-40.627,-53.339,174.889,16.799,152.602
C03103=1090.478,-40.388,-53.350,174.890,16.800,152.602
C03104=1090.483,-40.138,-53.363,174.892,16.801,152.602
C03105=1090.490,-39.888,-53.375,174.894,16.802,152.602
C03106=1090.495,-39.639,-53.387,174.896,16.805,152.602
C03107=1090.501,-39.389,-53.400,174.897,16.806,152.602
C03108=1090.508,-39.139,-53.411,174.899,16.807,152.602
C03109=1090.513,-38.890,-53.423,174.900,16.808,152.602
C03110=1090.519,-38.640,-53.436,174.902,16.810,152.602
C03111=1090.525,-38.390,-53.448,174.904,16.811,152.601
C03112=1090.531,-38.141,-53.460,174.905,16.812,152.602
C03113=1090.537,-37.891,-53.472,174.906,16.813,152.601
C03114=1090.543,-37.641,-53.485,174.908,16.814,152.601
C03115=1090.548,-37.392,-53.497,174.909,16.816,152.601
C03116=1090.554,-37.142,-53.510,174.912,16.818,152.601
C03117=1090.560,-36.893,-53.522,174.914,16.819,152.601
C03118=1090.566,-36.643,-53.534,174.915,16.821,152.601
C03119=1090.572,-36.394,-53.546,174.916,16.822,152.601
C03120=1090.578,-36.144,-53.559,174.918,16.823,152.601
C03121=1090.583,-35.895,-53.571,174.919,16.824,152.601
C03122=1090.589,-35.645,-53.584,174.921,16.825,152.601
C03123=1090.595,-35.395,-53.596,174.923,16.827,152.601
C03124=1090.601,-35.145,-53.608,174.924,16.828,152.601
C03125=1090.607,-34.896,-53.620,174.926,16.830,152.601
C03126=1090.613,-34.646,-53.633,174.928,16.831,152.601
C03127=1090.618,-34.396,-53.646,174.929,16.833,152.601
C03128=1090.624,-34.147,-53.658,174.931,16.834,152.601
C03129=1090.630,-33.897,-53.670,174.933,16.835,152.600
C03130=1090.636,-33.648,-53.682,174.934,16.836,152.600
C03131=1090.642,-33.398,-53.695,174.936,16.838,152.600
C03132=1090.649,-33.108,-53.709,174.938,16.840,152.600
C03133=1090.656,-32.818,-53.723,174.939,16.841,152.600
C03134=1090.662,-32.528,-53.738,174.942,16.843,152.600
C03135=1090.669,-32.238,-53.753,174.943,16.844,152.600
C03136=1090.674,-31.989,-53.765,174.945,16.845,152.600
C03137=1090.681,-31.739,-53.777,174.946,16.846,152.600
C03138=1090.687,-31.489,-53.790,174.949,16.849,152.600
C03139=1090.693,-31.239,-53.802,174.950,16.850,152.600
C03140=1090.699,-30.989,-53.815,174.952,16.851,152.600
C03141=1090.704,-30.741,-53.828,174.953,16.852,152.600
C03142=1090.710,-30.491,-53.840,174.955,16.854,152.600
C03143=1090.716,-30.241,-53.853,174.956,16.855,152.600
C03144=1090.722,-29.991,-53.865,174.958,16.856,152.600
C03145=1090.728,-29.741,-53.878,174.959,16.857,152.600
C03146=1090.733,-29.492,-53.890,174.962,16.860,152.600
C03147=1090.739,-29.242,-53.903,174.963,16.861,152.599
C03148=1090.746,-28.993,-53.915,174.965,16.862,152.599
C03149=1090.752,-28.743,-53.928,174.966,16.863,152.599
C03150=1090.758,-28.493,-53.940,174.968,16.865,152.599
C03151=1090.763,-28.244,-53.953,174.969,16.866,152.599
C03152=1090.769,-27.994,-53.965,174.971,16.867,152.599
C03153=1090.775,-27.745,-53.978,174.973,16.869,152.599
C03154=1090.781,-27.495,-53.991,174.975,16.870,152.599
C03155=1090.787,-27.245,-54.003,174.976,16.872,152.599
C03156=1090.793,-26.995,-54.016,174.978,16.873,152.599
C03157=1090.799,-26.747,-54.029,174.979,16.874,152.599
C03158=1090.805,-26.497,-54.041,174.981,16.876,152.599
C03159=1090.811,-26.247,-54.054,174.983,16.877,152.599
C03160=1090.816,-25.997,-54.067,174.985,16.879,152.599
C03161=1090.823,-25.748,-54.080,174.986,16.880,152.599
C03162=1090.828,-25.499,-54.092,174.988,16.881,152.599
C03163=1090.833,-25.249,-54.105,174.989,16.883,152.599
C03164=1090.839,-24.999,-54.118,174.991,16.884,152.599
C03165=1090.845,-24.749,-54.131,174.992,16.885,152.599
C03166=1090.851,-24.500,-54.144,174.995,16.887,152.598
C03167=1090.857,-24.250,-54.156,174.996,16.888,152.598
C03168=1090.863,-24.001,-54.169,174.998,16.890,152.598
C03169=1090.869,-23.751,-54.182,174.999,16.891,152.598
C03170=1090.875,-23.501,-54.194,175.001,16.893,152.598
C03171=1090.880,-23.252,-54.208,175.002,16.894,152.598
C03172=1090.886,-23.002,-54.221,175.005,16.895,152.598
C03173=1090.892,-22.752,-54.233,175.006,16.897,152.598
C03174=1090.897,-22.503,-54.246,175.008,16.898,152.598
C03175=1090.903,-22.254,-54.259,175.009,16.899,152.598
C03176=1090.909,-22.004,-54.271,175.011,16.901,152.598
C03177=1090.915,-21.754,-54.284,175.012,16.902,152.598
C03178=1090.921,-21.504,-54.298,175.014,16.904,152.598
C03179=1090.927,-21.255,-54.311,175.016,16.905,152.598
C03180=1090.933,-21.005,-54.323,175.018,16.906,152.598
C03181=1090.939,-20.755,-54.336,175.019,16.908,152.598
C03182=1090.944,-20.507,-54.349,175.021,16.909,152.598
C03183=1090.950,-20.257,-54.361,175.022,16.911,152.598
C03184=1090.956,-20.007,-54.375,175.024,16.912,152.598
C03185=1090.962,-19.757,-54.388,175.026,16.914,152.597
C03186=1090.968,-19.508,-54.401,175.027,16.915,152.597
C03187=1090.974,-19.258,-54.414,175.029,16.916,152.597
C03188=1090.980,-19.009,-54.427,175.031,16.917,152.597
C03189=1090.985,-18.759,-54.440,175.033,16.920,152.597
C03190=1090.991,-18.509,-54.453,175.034,16.921,152.597
C03191=1090.997,-18.260,-54.466,175.036,16.922,152.597
C03192=1091.003,-18.010,-54.478,175.037,16.923,152.597
C03193=1091.009,-17.760,-54.492,175.039,16.925,152.597
C03194=1091.014,-17.511,-54.504,175.040,16.926,152.597
C03195=1091.020,-17.262,-54.518,175.043,16.928,152.597
C03196=1091.027,-16.991,-54.532,175.044,16.929,152.597
C03197=1091.033,-16.720,-54.546,175.046,16.931,152.597
C03198=1091.039,-16.448,-54.560,175.048,16.932,152.597
C03199=1091.046,-16.177,-54.574,175.049,16.934,152.597
C03200=1091.052,-15.928,-54.588,175.051,16.935,152.597
C03201=1091.058,-15.678,-54.600,175.054,16.937,152.597
C03202=1091.064,-15.429,-54.613,175.055,16.938,152.597
C03203=1091.070,-15.179,-54.627,175.057,16.939,152.596
C03204=1091.076,-14.929,-54.640,175.058,16.940,152.596
C03205=1091.082,-14.680,-54.653,175.060,16.942,152.596
C03206=1091.087,-14.430,-54.666,175.062,16.944,152.596
C03207=1091.093,-14.181,-54.680,175.063,16.945,152.596
C03208=1091.099,-13.931,-54.693,175.065,16.946,152.596
C03209=1091.105,-13.681,-54.706,175.066,16.948,152.596
C03210=1091.110,-13.433,-54.719,175.068,16.949,152.596
C03211=1091.115,-13.183,-54.732,175.070,16.951,152.596
C03212=1091.122,-12.933,-54.745,175.072,16.953,152.596
C03213=1091.127,-12.684,-54.759,175.073,16.954,152.596
C03214=1091.133,-12.434,-54.772,175.075,16.955,152.596
C03215=1091.139,-12.185,-54.785,175.076,16.956,152.596
C03216=1091.145,-11.935,-54.799,175.078,16.959,152.596
C03217=1091.151,-11.685,-54.811,175.080,16.960,152.596
C03218=1091.156,-11.435,-54.825,175.082,16.961,152.596
C03219=1091.162,-11.186,-54.839,175.083,16.962,152.596
C03220=1091.167,-10.936,-54.852,175.085,16.963,152.596
C03221=1091.174,-10.687,-54.865,175.087,16.966,152.596
C03222=1091.180,-10.438,-54.878,175.088,16.967,152.596
C03223=1091.185,-10.188,-54.892,175.090,16.968,152.596
C03224=1091.191,-9.938,-54.905,175.091,16.970,152.596
C03225=1091.197,-9.688,-54.918,175.094,16.971,152.595
C03226=1091.203,-9.439,-54.932,175.095,16.973,152.595
C03227=1091.208,-9.189,-54.945,175.097,16.974,152.595
C03228=1091.214,-8.940,-54.958,175.098,16.975,152.595
C03229=1091.220,-8.690,-54.972,175.100,16.977,152.595
C03230=1091.226,-8.441,-54.985,175.102,16.978,152.595
C03231=1091.232,-8.192,-54.999,175.104,16.979,152.595
C03232=1091.238,-7.941,-55.012,175.105,16.981,152.595
C03233=1091.244,-7.691,-55.025,175.107,16.982,152.595
C03234=1091.250,-7.442,-55.039,175.109,16.984,152.595
C03235=1091.256,-7.193,-55.053,175.111,16.985,152.595
C03236=1091.261,-6.943,-55.066,175.112,16.987,152.595
C03237=1091.267,-6.693,-55.079,175.114,16.988,152.595
C03238=1091.273,-6.444,-55.093,175.115,16.989,152.595
C03239=1091.279,-6.194,-55.106,175.118,16.991,152.595
C03240=1091.284,-5.945,-55.120,175.119,16.993,152.595
C03241=1091.291,-5.696,-55.133,175.121,16.994,152.595
C03242=1091.296,-5.446,-55.147,175.122,16.995,152.595
C03243=1091.302,-5.197,-55.160,175.124,16.997,152.595
C03244=1091.308,-4.946,-55.173,175.126,16.998,152.594
C03245=1091.314,-4.697,-55.187,175.127,17.000,152.594
C03246=1091.320,-4.447,-55.201,175.129,17.001,152.594
C03247=1091.326,-4.198,-55.214,175.131,17.003,152.594
C03248=1091.332,-3.948,-55.228,175.133,17.004,152.594
C03249=1091.338,-3.699,-55.241,175.134,17.005,152.594
C03250=1091.343,-3.449,-55.255,175.136,17.006,152.594
C03251=1091.349,-3.200,-55.269,175.138,17.009,152.594
C03252=1091.355,-2.950,-55.282,175.140,17.010,152.594
C03253=1091.360,-2.701,-55.296,175.141,17.011,152.594
C03254=1091.366,-2.451,-55.310,175.143,17.012,152.594
C03255=1091.372,-2.201,-55.323,175.145,17.014,152.594
C03256=1091.378,-1.951,-55.337,175.147,17.016,152.594
C03257=1091.383,-1.702,-55.351,175.148,17.017,152.594
C03258=1091.389,-1.452,-55.365,175.150,17.018,152.594
C03259=1091.395,-1.203,-55.378,175.152,17.020,152.594
C03260=1091.401,-0.930,-55.393,175.153,17.022,152.594
C03261=1091.407,-0.658,-55.408,175.155,17.023,152.594
C03262=1091.413,-0.385,-55.424,175.157,17.025,152.594
C03263=1091.420,-0.113,-55.439,175.159,17.026,152.594
C03264=1091.425,0.137,-55.452,175.161,17.028,152.593
C03265=1091.431,0.386,-55.466,175.163,17.029,152.593
C03266=1091.437,0.636,-55.480,175.164,17.030,152.593
C03267=1091.442,0.885,-55.493,175.166,17.032,152.593
C03268=1091.448,1.135,-55.507,175.168,17.034,152.593
C03269=1091.454,1.385,-55.522,175.170,17.035,152.593
C03270=1091.460,1.635,-55.535,175.171,17.037,152.593
C03271=1091.466,1.884,-55.549,175.173,17.038,152.593
C03272=1091.471,2.134,-55.563,175.175,17.040,152.593
C03273=1091.477,2.383,-55.576,175.176,17.041,152.593
C03274=1091.483,2.633,-55.590,175.178,17.042,152.593
C03275=1091.488,2.882,-55.604,175.180,17.044,152.593
C03276=1091.495,3.132,-55.618,175.182,17.045,152.593
C03277=1091.500,3.381,-55.632,175.183,17.047,152.593
C03278=1091.506,3.631,-55.646,175.185,17.048,152.593
C03279=1091.512,3.880,-55.659,175.187,17.050,152.593
C03280=1091.517,4.130,-55.673,175.189,17.051,152.593
C03281=1091.523,4.379,-55.687,175.190,17.052,152.593
C03282=1091.529,4.630,-55.701,175.192,17.054,152.592
C03283=1091.535,4.879,-55.716,175.194,17.056,152.592
C03284=1091.541,5.128,-55.729,175.196,17.057,152.592
C03285=1091.546,5.377,-55.743,175.197,17.058,152.592
C03286=1091.552,5.627,-55.757,175.199,17.060,152.592
C03287=1091.558,5.877,-55.771,175.201,17.061,152.592
C03288=1091.564,6.126,-55.786,175.202,17.063,152.592
C03289=1091.569,6.376,-55.800,175.204,17.064,152.592
C03290=1091.575,6.625,-55.814,175.206,17.066,152.592
C03291=1091.581,6.875,-55.827,175.208,17.067,152.592
C03292=1091.587,7.125,-55.841,175.209,17.068,152.592
C03293=1091.593,7.374,-55.856,175.211,17.069,152.592
C03294=1091.598,7.623,-55.869,175.213,17.072,152.592
C03295=1091.604,7.873,-55.883,175.215,17.073,152.592
C03296=1091.610,8.123,-55.898,175.217,17.074,152.592
C03297=1091.616,8.372,-55.912,175.219,17.076,152.592
C03298=1091.622,8.622,-55.925,175.220,17.077,152.592
C03299=1091.627,8.871,-55.939,175.222,17.078,152.592
C03300=1091.634,9.121,-55.954,175.223,17.080,152.592
C03301=1091.639,9.370,-55.968,175.226,17.082,152.591
C03302=1091.645,9.620,-55.982,175.227,17.083,152.591
C03303=1091.651,9.870,-55.997,175.229,17.084,152.591
C03304=1091.656,10.119,-56.011,175.231,17.086,152.591
C03305=1091.662,10.369,-56.025,175.233,17.087,152.591
C03306=1091.668,10.617,-56.039,175.234,17.088,152.591
C03307=1091.674,10.868,-56.053,175.236,17.090,152.591
C03308=1091.680,11.117,-56.067,175.238,17.092,152.591
C03309=1091.686,11.366,-56.081,175.240,17.093,152.591
C03310=1091.692,11.616,-56.096,175.241,17.094,152.591
C03311=1091.697,11.866,-56.109,175.244,17.096,152.591
C03312=1091.703,12.115,-56.124,175.245,17.097,152.591
C03313=1091.709,12.365,-56.138,175.247,17.098,152.591
C03314=1091.715,12.614,-56.153,175.248,17.100,152.591
C03315=1091.720,12.864,-56.167,175.251,17.101,152.590
C03316=1091.727,13.113,-56.182,175.252,17.103,152.590
C03317=1091.732,13.363,-56.195,175.254,17.104,152.590
C03318=1091.738,13.613,-56.209,175.256,17.106,152.590
C03319=1091.745,13.862,-56.224,175.258,17.107,152.590
C03320=1091.750,14.111,-56.238,175.259,17.108,152.590
C03321=1091.756,14.360,-56.252,175.262,17.110,152.590
C03322=1091.762,14.611,-56.266,175.263,17.111,152.590
C03323=1091.767,14.860,-56.282,175.265,17.112,152.590
C03324=1091.774,15.134,-56.297,175.267,17.114,152.590
C03325=1091.781,15.409,-56.313,175.269,17.116,152.590
C03326=1091.786,15.684,-56.329,175.271,17.117,152.590
C03327=1091.793,15.958,-56.344,175.273,17.119,152.590
C03328=1091.799,16.208,-56.358,175.275,17.121,152.590
C03329=1091.804,16.457,-56.374,175.276,17.122,152.590
C03330=1091.810,16.707,-56.388,175.278,17.123,152.589
C03331=1091.815,16.956,-56.402,175.280,17.125,152.589
C03332=1091.822,17.206,-56.417,175.282,17.126,152.589
C03333=1091.827,17.455,-56.431,175.283,17.127,152.589
C03334=1091.833,17.705,-56.445,175.286,17.129,152.589
C03335=1091.839,17.954,-56.460,175.287,17.131,152.589
C03336=1091.845,18.203,-56.474,175.289,17.132,152.589
C03337=1091.850,18.454,-56.489,175.291,17.133,152.589
C03338=1091.856,18.703,-56.504,175.293,17.135,152.589
C03339=1091.862,18.953,-56.518,175.294,17.136,152.589
C03340=1091.868,19.202,-56.533,175.296,17.137,152.589
C03341=1091.874,19.451,-56.547,175.298,17.139,152.589
C03342=1091.879,19.701,-56.561,175.300,17.141,152.589
C03343=1091.885,19.951,-56.577,175.301,17.142,152.589
C03344=1091.890,20.200,-56.591,175.304,17.143,152.588
C03345=1091.897,20.450,-56.605,175.305,17.144,152.588
C03346=1091.902,20.699,-56.620,175.307,17.146,152.588
C03347=1091.908,20.948,-56.634,175.309,17.148,152.588
C03348=1091.914,21.198,-56.649,175.311,17.149,152.588
C03349=1091.919,21.447,-56.664,175.313,17.150,152.588
C03350=1091.925,21.698,-56.678,175.315,17.152,152.588
C03351=1091.931,21.947,-56.693,175.316,17.153,152.588
C03352=1091.936,22.196,-56.708,175.318,17.154,152.588
C03353=1091.943,22.446,-56.723,175.320,17.156,152.588
C03354=1091.948,22.695,-56.737,175.322,17.158,152.588
C03355=1091.954,22.945,-56.752,175.323,17.159,152.588
C03356=1091.960,23.194,-56.767,175.326,17.160,152.588
C03357=1091.965,23.444,-56.781,175.327,17.162,152.587
C03358=1091.971,23.693,-56.796,175.329,17.163,152.588
C03359=1091.976,23.943,-56.811,175.331,17.165,152.587
C03360=1091.983,24.192,-56.826,175.333,17.166,152.587
C03361=1091.989,24.441,-56.840,175.334,17.167,152.587
C03362=1091.994,24.692,-56.855,175.337,17.169,152.587
C03363=1092.000,24.941,-56.870,175.338,17.170,152.587
C03364=1092.006,25.190,-56.885,175.340,17.171,152.587
C03365=1092.011,25.440,-56.900,175.342,17.173,152.587
C03366=1092.017,25.689,-56.915,175.344,17.174,152.587
C03367=1092.023,25.939,-56.929,175.345,17.176,152.587
C03368=1092.029,26.188,-56.943,175.348,17.177,152.587
C03369=1092.034,26.438,-56.959,175.349,17.179,152.587
C03370=1092.040,26.687,-56.974,175.352,17.180,152.586
C03371=1092.047,26.936,-56.988,175.353,17.181,152.586
C03372=1092.052,27.186,-57.004,175.355,17.183,152.586
C03373=1092.058,27.436,-57.018,175.357,17.185,152.586
C03374=1092.063,27.685,-57.033,175.359,17.186,152.586
C03375=1092.069,27.935,-57.048,175.361,17.187,152.586
C03376=1092.075,28.184,-57.063,175.363,17.189,152.586
C03377=1092.081,28.434,-57.078,175.364,17.190,152.586
C03378=1092.086,28.683,-57.093,175.366,17.191,152.586
C03379=1092.092,28.933,-57.108,175.368,17.193,152.586
C03380=1092.098,29.182,-57.123,175.370,17.194,152.586
C03381=1092.103,29.432,-57.138,175.372,17.195,152.586
C03382=1092.109,29.681,-57.153,175.374,17.197,152.586
C03383=1092.116,29.930,-57.168,175.375,17.198,152.586
C03384=1092.121,30.180,-57.183,175.378,17.200,152.585
C03385=1092.127,30.430,-57.197,175.380,17.201,152.585
C03386=1092.132,30.679,-57.212,175.381,17.202,152.585
C03387=1092.138,30.929,-57.227,175.384,17.204,152.585
C03388=1092.144,31.204,-57.245,175.385,17.206,152.585
C03389=1092.150,31.480,-57.261,175.387,17.207,152.585
C03390=1092.156,31.757,-57.278,175.389,17.208,152.585
C03391=1092.163,32.032,-57.294,175.392,17.210,152.585
C03392=1092.169,32.282,-57.310,175.393,17.211,152.585
C03393=1092.174,32.531,-57.325,175.395,17.213,152.585
C03394=1092.180,32.781,-57.340,175.397,17.215,152.585
C03395=1092.186,33.030,-57.355,175.399,17.216,152.584
C03396=1092.191,33.280,-57.370,175.401,17.217,152.584
C03397=1092.197,33.529,-57.385,175.403,17.218,152.584
C03398=1092.203,33.779,-57.400,175.405,17.220,152.584
C03399=1092.210,34.028,-57.416,175.407,17.221,152.584
C03400=1092.215,34.277,-57.431,175.408,17.223,152.584
C03401=1092.221,34.527,-57.446,175.411,17.224,152.584
C03402=1092.226,34.776,-57.461,175.412,17.226,152.584
C03403=1092.232,35.026,-57.477,175.415,17.227,152.584
C03404=1092.237,35.275,-57.491,175.416,17.228,152.584
C03405=1092.243,35.525,-57.507,175.418,17.230,152.583
C03406=1092.250,35.775,-57.522,175.420,17.231,152.583
C03407=1092.255,36.024,-57.538,175.422,17.232,152.583
C03408=1092.261,36.273,-57.553,175.424,17.233,152.583
C03409=1092.266,36.523,-57.568,175.426,17.235,152.583
C03410=1092.272,36.772,-57.583,175.427,17.237,152.583
C03411=1092.278,37.022,-57.598,175.430,17.238,152.583
C03412=1092.283,37.271,-57.614,175.431,17.239,152.583
C03413=1092.290,37.520,-57.629,175.433,17.241,152.583
C03414=1092.296,37.770,-57.645,175.436,17.242,152.583
C03415=1092.301,38.020,-57.660,175.437,17.243,152.583
C03416=1092.307,38.269,-57.675,175.440,17.245,152.582
C03417=1092.312,38.519,-57.690,175.441,17.246,152.582
C03418=1092.318,38.768,-57.706,175.443,17.247,152.582
C03419=1092.324,39.018,-57.722,175.445,17.249,152.582
C03420=1092.330,39.267,-57.736,175.447,17.250,152.582
C03421=1092.335,39.517,-57.752,175.449,17.252,152.582
C03422=1092.341,39.765,-57.768,175.451,17.253,152.582
C03423=1092.346,40.015,-57.783,175.452,17.254,152.582
C03424=1092.353,40.265,-57.798,175.455,17.256,152.582
C03425=1092.358,40.514,-57.814,175.456,17.257,152.582
C03426=1092.364,40.764,-57.830,175.459,17.259,152.581
C03427=1092.369,41.014,-57.845,175.461,17.260,152.581
C03428=1092.375,41.263,-57.860,175.462,17.261,152.581
C03429=1092.381,41.512,-57.876,175.465,17.263,152.581
C03430=1092.387,41.762,-57.892,175.466,17.264,152.581
C03431=1092.392,42.011,-57.907,175.469,17.266,152.581
C03432=1092.398,42.260,-57.923,175.470,17.267,152.581
C03433=1092.404,42.510,-57.938,175.472,17.268,152.581
C03434=1092.409,42.760,-57.953,175.474,17.270,152.581
C03435=1092.415,43.009,-57.969,175.476,17.271,152.580
C03436=1092.421,43.259,-57.985,175.478,17.272,152.580
C03437=1092.427,43.507,-58.000,175.480,17.273,152.580
C03438=1092.432,43.757,-58.016,175.482,17.275,152.580
C03439=1092.438,44.007,-58.031,175.484,17.276,152.580
C03440=1092.443,44.256,-58.047,175.486,17.278,152.580
C03441=1092.449,44.506,-58.063,175.488,17.279,152.580
C03442=1092.455,44.755,-58.079,175.490,17.281,152.580
C03443=1092.460,45.004,-58.094,175.492,17.282,152.580
C03444=1092.466,45.254,-58.110,175.494,17.283,152.580
C03445=1092.472,45.504,-58.126,175.495,17.284,152.579
C03446=1092.477,45.753,-58.141,175.498,17.286,152.579
C03447=1092.483,46.002,-58.158,175.499,17.287,152.579
C03448=1092.488,46.252,-58.173,175.502,17.289,152.579
C03449=1092.494,46.501,-58.189,175.503,17.290,152.579
C03450=1092.499,46.751,-58.204,175.505,17.291,152.579
C03451=1092.505,47.000,-58.221,175.508,17.293,152.579
C03452=1092.511,47.276,-58.238,175.510,17.295,152.579
C03453=1092.517,47.552,-58.255,175.512,17.296,152.579
C03454=1092.523,47.828,-58.273,175.514,17.297,152.578
C03455=1092.530,48.104,-58.291,175.516,17.299,152.578
C03456=1092.535,48.354,-58.306,175.518,17.300,152.578
C03457=1092.541,48.603,-58.322,175.521,17.302,152.578
C03458=1092.546,48.853,-58.338,175.522,17.303,152.578
C03459=1092.552,49.102,-58.354,175.524,17.304,152.578
C03460=1092.558,49.352,-58.369,175.526,17.306,152.578
C03461=1092.563,49.601,-58.385,175.528,17.307,152.578
C03462=1092.569,49.850,-58.402,175.530,17.308,152.578
C03463=1092.575,50.100,-58.417,175.532,17.310,152.577
C03464=1092.581,50.349,-58.433,175.534,17.311,152.577
C03465=1092.586,50.598,-58.449,175.536,17.312,152.577
C03466=1092.592,50.848,-58.465,175.538,17.313,152.577
C03467=1092.598,51.097,-58.481,175.540,17.315,152.577
C03468=1092.603,51.347,-58.497,175.542,17.316,152.577
C03469=1092.609,51.596,-58.513,175.544,17.318,152.577
C03470=1092.615,51.845,-58.529,175.546,17.319,152.577
C03471=1092.620,52.095,-58.544,175.548,17.321,152.577
C03472=1092.626,52.344,-58.561,175.550,17.321,152.576
C03473=1092.632,52.594,-58.577,175.553,17.323,152.576
C03474=1092.637,52.843,-58.592,175.554,17.324,152.576
C03475=1092.643,53.092,-58.608,175.556,17.325,152.576
C03476=1092.649,53.342,-58.625,175.558,17.327,152.576
C03477=1092.654,53.592,-58.641,175.560,17.328,152.576
C03478=1092.660,53.841,-58.657,175.562,17.330,152.576
C03479=1092.666,54.091,-58.673,175.564,17.331,152.576
C03480=1092.671,54.339,-58.689,175.567,17.332,152.575
C03481=1092.677,54.589,-58.705,175.568,17.333,152.575
C03482=1092.683,54.839,-58.721,175.571,17.335,152.575
C03483=1092.689,55.088,-58.737,175.573,17.336,152.575
C03484=1092.695,55.337,-58.753,175.574,17.337,152.575
C03485=1092.701,55.587,-58.770,175.577,17.339,152.575
C03486=1092.706,55.836,-58.785,175.578,17.340,152.575
C03487=1092.711,56.086,-58.802,175.581,17.341,152.574
C03488=1092.717,56.335,-58.818,175.583,17.342,152.574
C03489=1092.723,56.584,-58.834,175.585,17.344,152.574
C03490=1092.729,56.834,-58.850,175.587,17.345,152.574
C03491=1092.735,57.084,-58.866,175.589,17.347,152.574
C03492=1092.741,57.333,-58.882,175.591,17.348,152.574
C03493=1092.746,57.582,-58.898,175.593,17.348,152.574
C03494=1092.752,57.832,-58.915,175.595,17.350,152.573
C03495=1092.757,58.081,-58.931,175.597,17.351,152.573
C03496=1092.763,58.330,-58.947,175.599,17.353,152.573
C03497=1092.769,58.579,-58.964,175.601,17.353,152.573
C03498=1092.775,58.829,-58.980,175.604,17.355,152.573
C03499=1092.781,59.079,-58.996,175.605,17.356,152.573
C03500=1092.786,59.328,-59.012,175.608,17.358,152.573
C03501=1092.792,59.578,-59.029,175.609,17.359,152.572
C03502=1092.798,59.827,-59.045,175.612,17.360,152.572
C03503=1092.804,60.076,-59.061,175.614,17.361,152.572
C03504=1092.810,60.326,-59.077,175.616,17.363,152.572
C03505=1092.815,60.575,-59.094,175.618,17.364,152.572
C03506=1092.821,60.825,-59.111,175.620,17.365,152.572
C03507=1092.827,61.074,-59.127,175.622,17.366,152.571
C03508=1092.833,61.323,-59.143,175.624,17.367,152.571
C03509=1092.839,61.573,-59.159,175.626,17.369,152.571
C03510=1092.845,61.822,-59.176,175.628,17.370,152.571
C03511=1092.850,62.072,-59.192,175.630,17.371,152.571
C03512=1092.856,62.321,-59.209,175.632,17.372,152.571
C03513=1092.862,62.571,-59.225,175.635,17.374,152.570
C03514=1092.868,62.820,-59.241,175.636,17.375,152.570
C03515=1092.873,63.070,-59.258,175.639,17.376,152.570
C03516=1092.879,63.345,-59.276,175.641,17.377,152.570
C03517=1092.886,63.621,-59.294,175.643,17.379,152.570
C03518=1092.892,63.896,-59.312,175.646,17.380,152.570
C03519=1092.899,64.172,-59.331,175.648,17.382,152.569
C03520=1092.905,64.422,-59.347,175.650,17.382,152.569
C03521=1092.910,64.671,-59.364,175.653,17.384,152.569
C03522=1092.916,64.921,-59.380,175.654,17.385,152.569
C03523=1092.921,65.170,-59.397,175.657,17.386,152.569
C03524=1092.927,65.420,-59.413,175.659,17.387,152.569
C03525=1092.933,65.668,-59.430,175.660,17.388,152.569
C03526=1092.939,65.918,-59.447,175.663,17.390,152.568
C03527=1092.945,66.167,-59.463,175.665,17.391,152.568
C03528=1092.950,66.417,-59.480,175.667,17.392,152.568
C03529=1092.956,66.666,-59.496,175.669,17.394,152.568
C03530=1092.962,66.916,-59.512,175.672,17.395,152.568
C03531=1092.967,67.165,-59.530,175.673,17.396,152.568
C03532=1092.973,67.414,-59.546,175.676,17.398,152.567
C03533=1092.978,67.664,-59.563,175.678,17.398,152.567
C03534=1092.984,67.913,-59.579,175.680,17.400,152.567
C03535=1092.990,68.163,-59.596,175.682,17.400,152.567
C03536=1092.996,68.411,-59.613,175.684,17.402,152.567
C03537=1093.001,68.661,-59.630,175.686,17.403,152.567
C03538=1093.007,68.910,-59.646,175.689,17.404,152.566
C03539=1093.012,69.160,-59.663,175.690,17.406,152.566
C03540=1093.018,69.409,-59.680,175.693,17.407,152.566
C03541=1093.024,69.658,-59.697,175.695,17.408,152.566
C03542=1093.030,69.908,-59.713,175.697,17.409,152.566
C03543=1093.035,70.157,-59.730,175.699,17.410,152.565
C03544=1093.041,70.406,-59.747,175.701,17.412,152.565
C03545=1093.046,70.656,-59.764,175.703,17.413,152.565
C03546=1093.052,70.905,-59.780,175.706,17.414,152.565
C03547=1093.058,71.155,-59.798,175.707,17.415,152.565
C03548=1093.064,71.405,-59.815,175.710,17.416,152.565
C03549=1093.069,71.654,-59.831,175.712,17.418,152.565
C03550=1093.075,71.903,-59.849,175.714,17.419,152.564
C03551=1093.081,72.152,-59.865,175.716,17.420,152.564
C03552=1093.086,72.402,-59.882,175.719,17.421,152.564
C03553=1093.092,72.651,-59.899,175.721,17.422,152.564
C03554=1093.098,72.900,-59.916,175.723,17.424,152.564
C03555=1093.103,73.149,-59.933,175.725,17.425,152.564
C03556=1093.109,73.399,-59.950,175.727,17.426,152.563
C03557=1093.114,73.648,-59.966,175.729,17.427,152.563
C03558=1093.120,73.897,-59.984,175.732,17.428,152.563
C03559=1093.126,74.147,-60.000,175.733,17.429,152.563
C03560=1093.132,74.397,-60.018,175.736,17.431,152.563
C03561=1093.137,74.646,-60.035,175.738,17.432,152.562
C03562=1093.143,74.896,-60.051,175.740,17.433,152.562
C03563=1093.149,75.145,-60.069,175.743,17.435,152.562
C03564=1093.154,75.394,-60.086,175.745,17.435,152.562
C03565=1093.160,75.643,-60.103,175.747,17.437,152.562
C03566=1093.165,75.893,-60.119,175.749,17.438,152.561
C03567=1093.171,76.142,-60.137,175.752,17.439,152.561
C03568=1093.177,76.392,-60.154,175.753,17.440,152.561
C03569=1093.183,76.641,-60.171,175.756,17.442,152.561
C03570=1093.188,76.890,-60.188,175.758,17.442,152.561
C03571=1093.194,77.139,-60.205,175.760,17.444,152.561
C03572=1093.200,77.389,-60.222,175.762,17.444,152.560
C03573=1093.205,77.638,-60.239,175.765,17.446,152.560
C03574=1093.211,77.888,-60.257,175.767,17.447,152.560
C03575=1093.217,78.137,-60.274,175.769,17.448,152.560
C03576=1093.223,78.386,-60.291,175.771,17.449,152.560
C03577=1093.228,78.636,-60.308,175.774,17.450,152.559
C03578=1093.233,78.885,-60.326,175.775,17.451,152.559
C03579=1093.239,79.134,-60.342,175.778,17.453,152.559
C03580=1093.246,79.410,-60.361,175.780,17.454,152.559
C03581=1093.252,79.685,-60.381,175.782,17.455,152.559
C03582=1093.258,79.961,-60.400,175.785,17.457,152.558
C03583=1093.264,80.237,-60.419,175.788,17.458,152.558
C03584=1093.269,80.486,-60.436,175.790,17.459,152.558
C03585=1093.275,80.736,-60.454,175.792,17.460,152.558
C03586=1093.282,80.985,-60.471,175.795,17.461,152.557
C03587=1093.287,81.235,-60.488,175.796,17.462,152.557
C03588=1093.292,81.484,-60.505,175.799,17.464,152.557
C03589=1093.298,81.733,-60.523,175.801,17.465,152.557
C03590=1093.304,81.983,-60.540,175.803,17.466,152.557
C03591=1093.309,82.232,-60.558,175.805,17.466,152.557
C03592=1093.315,82.481,-60.575,175.808,17.468,152.556
C03593=1093.320,82.731,-60.592,175.810,17.469,152.556
C03594=1093.325,82.980,-60.610,175.812,17.470,152.556
C03595=1093.332,83.229,-60.627,175.815,17.472,152.556
C03596=1093.338,83.478,-60.645,175.817,17.472,152.555
C03597=1093.343,83.728,-60.662,175.819,17.474,152.555
C03598=1093.349,83.977,-60.679,175.821,17.475,152.555
C03599=1093.355,84.227,-60.697,175.824,17.476,152.555
C03600=1093.360,84.476,-60.715,175.825,17.477,152.555
C03601=1093.366,84.725,-60.732,175.828,17.478,152.554
C03602=1093.371,84.974,-60.749,175.830,17.479,152.554
C03603=1093.377,85.224,-60.767,175.832,17.480,152.554
C03604=1093.383,85.473,-60.785,175.834,17.481,152.554
C03605=1093.388,85.722,-60.802,175.837,17.482,152.554
C03606=1093.394,85.971,-60.820,175.839,17.484,152.553
C03607=1093.400,86.221,-60.838,175.841,17.484,152.553
C03608=1093.405,86.471,-60.854,175.844,17.486,152.553
C03609=1093.410,86.720,-60.872,175.846,17.487,152.553
C03610=1093.417,86.970,-60.890,175.848,17.488,152.553
C03611=1093.422,87.219,-60.908,175.850,17.489,152.552
C03612=1093.428,87.468,-60.925,175.853,17.490,152.552
C03613=1093.434,87.717,-60.943,175.855,17.491,152.552
C03614=1093.439,87.966,-60.961,175.857,17.492,152.552
C03615=1093.445,88.215,-60.978,175.860,17.493,152.551
C03616=1093.451,88.465,-60.996,175.862,17.494,152.551
C03617=1093.456,88.714,-61.014,175.865,17.496,152.551
C03618=1093.462,88.963,-61.031,175.866,17.496,152.551
C03619=1093.468,89.214,-61.048,175.869,17.497,152.551
C03620=1093.473,89.463,-61.066,175.871,17.498,152.550
C03621=1093.479,89.712,-61.084,175.874,17.499,152.550
C03622=1093.485,89.961,-61.102,175.875,17.500,152.550
C03623=1093.490,90.210,-61.119,175.878,17.502,152.550
C03624=1093.496,90.460,-61.137,175.881,17.503,152.549
C03625=1093.502,90.709,-61.155,175.883,17.503,152.549
C03626=1093.508,90.958,-61.172,175.886,17.505,152.549
C03627=1093.513,91.207,-61.190,175.887,17.505,152.549
C03628=1093.519,91.456,-61.208,175.890,17.507,152.548
C03629=1093.525,91.705,-61.226,175.892,17.507,152.548
C03630=1093.530,91.955,-61.244,175.894,17.509,152.548
C03631=1093.536,92.205,-61.262,175.897,17.510,152.548
C03632=1093.541,92.454,-61.280,175.899,17.511,152.548
